// TwinCAT 3 PLC project XtsLib
// Title: Xts Library
// Company: BeckhoffUK
// Author: ChrisK
// ProjectVersion: 1.0.0.6
// Description: Xts framework implementation
// ProgramVersion: 3.1.4023.0
// libraries:
//   Tc2_Standard, * (Beckhoff Automation GmbH)
//   Tc2_System, * (Beckhoff Automation GmbH)
//   Tc3_EventLogger, * (Beckhoff Automation GmbH)
//   Tc3_McCoordinatedMotion, * (Beckhoff Automation GmbH)
//   Tc3_Module, * (Beckhoff Automation GmbH)
//   Tc3_PackML_V2, * (Beckhoff Automation GmbH)
//   Tc3_XTS_Utility, * (Beckhoff Automation GmbH)
//   Tc2_MC2,newest,Beckhoff Automation GmbH
//   Tc3_Mc3Definitions,newest,Beckhoff Automation GmbH
//   Tc3_McCollisionAvoidance,newest,Beckhoff Automation GmbH
// project tree:
//   Axis Class/ MC2_Axis_Base.TcPOU
//   EventLoggerClass/ ITcMessage_Ext.TcIO, TcMessage_Ext.TcPOU
//   Mover Class/ FB_Mover.TcPOU, GearMover.TcPOU, IDynamics.TcIO, IGearMover.TcIO, IMover.TcIO, ITmsMover.TcIO, TMS_Mover.TcPOU
//   PackML/ IPmlStateMachine.TcIO, PMLStateMachine.TcPOU
//   PackML_Method_Pattern/ PML_Method_Base.TcPOU
//   SequenceSamples/ GearMoverSequence.TcPOU (not stored), IndexMoverSequence.TcPOU, IndexSequenceState.TcDUT, MoverSequenceInfo.TcDUT
//   Station Class/Process/ IProcess.TcIO, Process.TcPOU
//   Station Class/Station/ IStation.TcIO, Station.TcPOU, StationSample.TcPOU, stStationInfo.TcDUT, stStationStatus.TcDUT
//   Station Class/TMSStation/ ITF_SwitchStation.TcIO, TmsEmbarkStation.TcPOU, TmsExchange.TcPOU, TmsHoldStation.TcPOU
//   Switch Class/ DualModuleTmsSwitch.TcPOU, ITF_TmsSwitch.TcIO, TmsSwitchPosition.TcDUT, TmsSwitchInfo.TcDUT, TmsSwitchMode.TcDUT, TmsSwitchState.TcDUT
//   / SystemParameters.TcGVL
//   Tasks/ ActivateTrackForMover.TcPOU, AddMoverToGroupTask.TcPOU, AxesReset.TcPOU, DisableGroup.TcPOU, EnableGroup.TcPOU, GearInCA.TcPOU, HaltMover.TcPOU, Mc2Halt.TcPOU, ITask.TcIO, Mc2MoveToPosition.TcPOU, MoveModuloMoverToPosition.TcPOU, MoveMoverToPosition.TcPOU, MoveMoverToPositionZoned.TcPOU, RemoveAllMoverFromGroup.TcPOU, ResetGroup.TcPOU, StopMoverGroup.TcPOU, XtsDisableSequence.TcPOU, XtsEnableSequence.TcPOU
//   XTS Class/ ITF_StartUpSequence.TcIO, IXtsTrack.TcIO, XtsTrack.TcPOU
//   XTS Class/Xts Collision Group/ CAGroupInfo.TcDUT (not stored), CAGroupStatus.TcDUT (not stored), CollisionGroup.TcPOU, ICollisionGroup.TcIO (not stored)
//   XTS Class/Xts Hardware/ XtsHardware.TcPOU, XtsHardwareInfo.TcDUT, XtsHardwareState.TcDUT

// ---- SequenceSamples/IndexSequenceState.TcDUT
{attribute 'qualified_only'}
{attribute 'strict'}
TYPE IndexSequenceState :
(
	Init := 0,                                               
	Available := 1,
	MovingToStart := 2, 
	AtStart := 3,                                 
	MovingToStation := 4,
	QueuedAtStation := 5,
	AtStation := 6,
	AtProcess := 7,
	InProcess := 8,
	GetNextMove := 9,
	GoToNextStation := 10,
	Stopping := 11,
	Aborting := 12
);
END_TYPE

// ---- SequenceSamples/MoverSequenceInfo.TcDUT
TYPE MoverSequenceInfo :
STRUCT
	MoverId : UDINT;
	CurrentStation : INT;
	Velocity : MC_LREAL;
	State : IndexSequenceState;
END_STRUCT
END_TYPE

// ---- Station Class/Station/stStationInfo.TcDUT
TYPE stStationInfo :
STRUCT
	StationProcessTime : TIME;
	StationPosition : MC_LREAL;
	StationStatus : stStationStatus;
END_STRUCT
END_TYPE

// ---- Station Class/Station/stStationStatus.TcDUT
TYPE stStationStatus :
STRUCT
	Clear : BOOL;
	Complete : BOOL;
	Operating : BOOL;
	Ready : BOOL;
	HasMover : BOOL;
END_STRUCT
END_TYPE

// ---- Switch Class/TmsSwitchPosition.TcDUT
{attribute 'qualified_only'}
{attribute 'strict'}
TYPE TmsSwitchPosition :
(
	Up := 0,
	Middle := 1,
	Down := 2,
	Moving := 3
);
END_TYPE

// ---- Switch Class/TmsSwitchInfo.TcDUT
TYPE TmsSwitchInfo :
STRUCT
	State : TmsSwitchState;
	Mode : TmsSwitchMode;
	Position : TmsSwitchPosition;
	ActPos : MC_LREAL;
END_STRUCT
END_TYPE

// ---- Switch Class/TmsSwitchMode.TcDUT
{attribute 'qualified_only'}
{attribute 'strict'}
TYPE TmsSwitchMode :
(
	Automatic := 0,
	Manual := 1
);
END_TYPE

// ---- Switch Class/TmsSwitchState.TcDUT
{attribute 'qualified_only'}
{attribute 'strict'}
TYPE TmsSwitchState :
(
	Init := 0,                                               
	Ready := 1,                                 
	Enabling := 2,
	Enabled := 3,
	Resetting := 4,
	Waiting := 5,
	AssignMover := 6,
	Moving := 7,
	Done := 8,
	Disabling := 9
);
END_TYPE

// ---- XTS Class/Xts Hardware/XtsHardwareInfo.TcDUT
TYPE XtsHardwareInfo :
STRUCT
	NoOfParts: UDINT;
	NoOfTracks : UDINT;
	NoOfModules : ARRAY[1..10] OF UDINT;
	HWState : XtsHardwareState;
END_STRUCT
END_TYPE

// ---- XTS Class/Xts Hardware/XtsHardwareState.TcDUT
{attribute 'qualified_only'}
{attribute 'strict'}
TYPE XtsHardwareState :
(
	Init := 0,
	SetDetection := 1,                                               
	Redetect := 2,
	MoversValid := 3,                                 
	AllMoversFound := 4,
	MoverIdDetection := 5,
	XTSMode := 6,
	CheckModuleVoltages := 7,
	HWReady := 8
);
END_TYPE

// ---- SystemParameters.TcGVL
{attribute 'qualified_only'}
VAR_GLOBAL CONSTANT
	nModuleNumber  : UINT := 16;
	NumberOfMovers : INT := 10;
	NumberOfStations : INT := 6;
	TrackLength : LREAL := 4000.0;
	TrackHomePosition : LREAL := 800.0;
	Tracks : UDINT := 1;
END_VAR

// ---- EventLoggerClass/ITcMessage_Ext.TcIO
INTERFACE ITcMessage_Ext

METHOD Send : BOOL
VAR_INPUT
	eventType : Tc3_EventLogger.TcEventEntry;
	args : STRING(255);
END_VAR
END_METHOD

END_INTERFACE

// ---- Mover Class/IDynamics.TcIO
INTERFACE IDynamics

PROPERTY Acceleration : mc_lreal
GET
END_GET
SET
END_SET
END_PROPERTY

PROPERTY Deceleration : mc_lreal
GET
END_GET
SET
END_SET
END_PROPERTY

PROPERTY Jerk : mc_lreal
GET
END_GET
SET
END_SET
END_PROPERTY

END_INTERFACE

// ---- Mover Class/IGearMover.TcIO
INTERFACE IGearMover EXTENDS IMover

METHOD Gear : BOOL
VAR_INPUT
	MasterPosition : MC_LREAL;
	SlavePosition : MC_LREAL;
END_VAR
END_METHOD

METHOD inGear : BOOL
VAR_INPUT
END_VAR
END_METHOD

METHOD isMaster : BOOL
VAR_INPUT
END_VAR
END_METHOD

METHOD masterAxis : UDINT
VAR_INPUT
END_VAR
END_METHOD

END_INTERFACE

// ---- Mover Class/IMover.TcIO
INTERFACE IMover EXTENDS __SYSTEM.IQueryInterface

PROPERTY AxisRef : reference to axis_ref
GET
END_GET
END_PROPERTY

METHOD DisableAxis : BOOL
VAR_INPUT
END_VAR
END_METHOD

METHOD EnableAxis : BOOL
VAR_INPUT
END_VAR
END_METHOD

METHOD HaltAxis : BOOL
VAR_INPUT
END_VAR
END_METHOD

METHOD HasCommand : BOOL
VAR_INPUT
END_VAR
END_METHOD

METHOD hasError : BOOL
VAR_INPUT
END_VAR
END_METHOD

PROPERTY IdentInGroup : int
GET
END_GET
SET
END_SET
END_PROPERTY

METHOD isAtPosition : BOOL
VAR_INPUT
	position : MC_LREAL;
END_VAR
END_METHOD

METHOD isDetected : BOOL
VAR_INPUT
END_VAR
END_METHOD

METHOD isEnabled : BOOL
VAR_INPUT
END_VAR
END_METHOD

METHOD isPastPosition : BOOL
VAR_INPUT
	position : MC_LREAL;
END_VAR
END_METHOD

METHOD isStationary : BOOL
VAR_INPUT
END_VAR
END_METHOD

METHOD MoveTo : BOOL
VAR_INPUT
	Position : MC_LREAL;
	Velocity : MC_LREAL;
	BackwardMove : BOOL;
END_VAR
END_METHOD

METHOD ResetAxis : BOOL
VAR_INPUT
END_VAR
END_METHOD

END_INTERFACE

// ---- Mover Class/ITmsMover.TcIO
INTERFACE ITmsMover EXTENDS IMover

METHOD ActivateTrack : BOOL
VAR_INPUT
	newTrack : OTCID;
END_VAR
END_METHOD

PROPERTY ActiveTrack : OTCID
GET
END_GET
END_PROPERTY

METHOD SetMoverInterface : BOOL
VAR_INPUT
	MoverInterface : I_TcIoXtsXpuMover;
END_VAR
END_METHOD

END_INTERFACE

// ---- PackML/IPmlStateMachine.TcIO
INTERFACE IPmlStateMachine

METHOD public GetCurrentMode : E_PmlProtectedUnitMode
VAR_INPUT
END_VAR
END_METHOD

METHOD GetCurrentState : E_PMLState
VAR_INPUT
END_VAR
END_METHOD

METHOD PmlModeCommand : BOOL
VAR_INPUT
	Mode : E_PMLProtectedUnitMode;
END_VAR
END_METHOD

METHOD PmlStateCommand : bool
VAR_INPUT
	Command : E_PMLCommand;
END_VAR
END_METHOD

METHOD SetStateComplete : BOOL
VAR_INPUT
END_VAR
END_METHOD

END_INTERFACE

// ---- Station Class/Process/IProcess.TcIO
INTERFACE IProcess EXTENDS IStation

PROPERTY EndPosition : MC_LREAL
GET
END_GET
SET
END_SET
END_PROPERTY

PROPERTY IsProcess : booL
GET
END_GET
SET
END_SET
END_PROPERTY

PROPERTY ProcessVelocity : mc_lreal
GET
END_GET
SET
END_SET
END_PROPERTY

PROPERTY StartPosition : MC_LREAL
GET
END_GET
SET
END_SET
END_PROPERTY

END_INTERFACE

// ---- Station Class/Station/IStation.TcIO
INTERFACE IStation

METHOD Abort : BOOL
VAR_INPUT
END_VAR
END_METHOD

METHOD HasMover : BOOL
VAR_INPUT
	mover : IMover;
END_VAR
END_METHOD

METHOD IsClear : BOOL
VAR_INPUT
END_VAR
END_METHOD

METHOD isComplete : BOOL
VAR_INPUT
END_VAR
END_METHOD

PROPERTY IsLastStation : BOOL
GET
END_GET
SET
END_SET
END_PROPERTY

METHOD IsOperating : BOOL
VAR_INPUT
END_VAR
END_METHOD

METHOD IsReady : BOOL
VAR_INPUT
END_VAR
END_METHOD

METHOD MoverAway : BOOL
VAR_INPUT
END_VAR
END_METHOD

PROPERTY Position : MC_LREAL
GET
END_GET
SET
END_SET
END_PROPERTY

END_INTERFACE

// ---- Station Class/TMSStation/ITF_SwitchStation.TcIO
INTERFACE ITF_SwitchStation EXTENDS __SYSTEM.IQueryInterface

PROPERTY StationPosition : int
GET
END_GET
SET
END_SET
END_PROPERTY

METHOD SwitchMoveComplete : BOOL
VAR_INPUT
END_VAR
END_METHOD

PROPERTY SwitchPosition : mc_lreal
GET
END_GET
SET
END_SET
END_PROPERTY

END_INTERFACE

// ---- Switch Class/ITF_TmsSwitch.TcIO
INTERFACE ITF_TmsSwitch

METHOD ExchangeMover : BOOL
VAR_INPUT
	Mover : IMover;
	currentStation : ITF_SwitchStation;
END_VAR
END_METHOD

METHOD HasMover : BOOL
VAR_INPUT
END_VAR
END_METHOD

METHOD IsStationary : BOOL
VAR_INPUT
END_VAR
END_METHOD

METHOD MoveTo : BOOL
VAR_INPUT
	positionState : TmsSwitchPosition;
END_VAR
END_METHOD

PROPERTY Switch : TmsSwitchPosition
GET
END_GET
END_PROPERTY

END_INTERFACE

// ---- Tasks/ITask.TcIO
INTERFACE ITask

METHOD Abort : BOOL
VAR_INPUT
END_VAR
END_METHOD

PROPERTY Busy : bool
GET
END_GET
END_PROPERTY

PROPERTY Done : bool
GET
END_GET
END_PROPERTY

PROPERTY Error : bool
GET
END_GET
END_PROPERTY

END_INTERFACE

// ---- XTS Class/ITF_StartUpSequence.TcIO
INTERFACE ITF_StartUpSequence

METHOD Call : BOOL
VAR_INPUT
END_VAR
END_METHOD

END_INTERFACE

// ---- XTS Class/IXtsTrack.TcIO
INTERFACE IXtsTrack

PROPERTY HomePosition : MC_LREAL
GET
END_GET
SET
END_SET
END_PROPERTY

PROPERTY TrackLength : mc_lreal
GET
END_GET
SET
END_SET
END_PROPERTY

END_INTERFACE

// ---- Axis Class/MC2_Axis_Base.TcPOU
FUNCTION_BLOCK MC2_Axis_Base EXTENDS CyclicBase
VAR_INPUT
END_VAR
VAR_OUTPUT
END_VAR
VAR
	_axis : Tc2_MC2.AXIS_REF;
	axesEnable		: AxisPower(_axis);
	axesReset		: AxesReset(_axis);
	axesMoveTo 		: Mc2MoveToPosition(_axis);
	axesHalt 		: Mc2Halt(_axis);
	axesReadError : Tc2_MC2.MC_ReadAxisError;
	_MoverErrorId: DWORD;
END_VAR

METHOD Cycle : BOOL
VAR_INPUT
END_VAR
axesMoveTo.Cycle();
axesHalt.Cycle();
axesReset.Cycle();
_axis.ReadStatus();
axesEnable.Cycle();
axesReadError(Axis := _axis, Enable := TRUE, AxisErrorID => _MoverErrorId);
END_METHOD

METHOD PUBLIC DisableAxis : BOOL
VAR_INPUT
END_VAR
DisableAxis := axesEnable.Disable();
END_METHOD

METHOD PUBLIC EnableAxis : BOOL
VAR_INPUT
END_VAR
EnableAxis := axesEnable.Enable();
END_METHOD

METHOD PUBLIC HaltAxis : BOOL
VAR_INPUT
END_VAR
IF NOT axesHalt.Busy THEN
	axesHalt.Execute();
	axesMoveTo.Abort();
	HaltAxis := TRUE;
END_IF
END_METHOD

METHOD hasError : BOOL
VAR_INPUT
END_VAR
hasError := _axis.Status.Error;
END_METHOD

METHOD isAtPosition : BOOL
VAR_INPUT
	position : MC_LREAL;
END_VAR
IF _axis.NcToPlc.ActPos < position + 0.2 AND _axis.NcToPlc.ActPos > position - 0.2 THEN
	isAtPosition := TRUE;
END_IF
END_METHOD

METHOD isEnabled : BOOL
VAR_INPUT
END_VAR
isEnabled := not _axis.Status.Disabled;
END_METHOD

METHOD PUBLIC isStationary : BOOL
VAR_INPUT
END_VAR
isStationary := _axis.NcToPlc.SetVelo = 0;
END_METHOD

METHOD PUBLIC MoveToPosition : BOOL
VAR_INPUT
	Position : MC_LREAL;
	Velocity : MC_LREAL;
END_VAR
IF NOT isAtPosition(position := Position) THEN
	IF NOT axesMoveTo.Busy THEN
		axesMoveTo.MoveTo(Position := Position, Velocity := Velocity);
		MoveToPosition := TRUE;
	END_IF
END_IF
END_METHOD

METHOD PUBLIC ResetAxis : BOOL
VAR_INPUT
END_VAR
axesReset.Execute();
axesMoveTo.Abort();
axesHalt.Abort();
END_METHOD

END_FUNCTION_BLOCK

// ---- Tasks/AxesReset.TcPOU
{attribute 'hide_all_locals'}
FUNCTION_BLOCK AxesReset EXTENDS TaskBase
VAR_INPUT
END_VAR
VAR_OUTPUT
END_VAR
VAR
	resetMover : Tc2_MC2.MC_Reset;
	_axis : REFERENCE TO Tc2_MC2.AXIS_REF;
	_ResetMover : BOOL;
END_VAR

METHOD Abort : BOOL
resetMover.Execute := FALSE;
_busy := FALSE;
_ResetMover := FALSE;
Abort := TRUE;
State := 0;
END_METHOD

METHOD Cycle : BOOL
VAR_INPUT
END_VAR
CASE State OF
	0:
		IF _ResetMover THEN
			_done := FALSE;
			_error := FALSE;
			_busy := TRUE;
			resetMover.Execute := TRUE;
			IF resetMover.Busy THEN
				State := 10;
				_ResetMover := FALSE;
			END_IF
		END_IF
	
	10:
		IF NOT resetMover.Busy THEN
			IF resetMover.Done THEN
				_done := TRUE;
			ELSIF resetMover.Error THEN
				_error := TRUE;
			END_IF
			_busy := FALSE;
			resetMover.Execute := FALSE;
			State := 0;
		END_IF
END_CASE

resetMover(Axis := _axis);
END_METHOD

METHOD Execute : BOOL
VAR_INPUT
END_VAR
Execute := _ResetMover := true;
END_METHOD

METHOD FB_init : BOOL
VAR_INPUT
	bInitRetains : BOOL; // if TRUE, the retain variables are initialized (warm start / cold start)
	bInCopyCode : BOOL;  // if TRUE, the instance afterwards gets moved into the copy code (online change)
	axis : reference TO AXIS_REF;
END_VAR
_axis REF= axis;
END_METHOD

END_FUNCTION_BLOCK

// ---- Tasks/Mc2MoveToPosition.TcPOU
FUNCTION_BLOCK Mc2MoveToPosition EXTENDS TaskBase
VAR_INPUT
END_VAR
VAR_OUTPUT
END_VAR
VAR
	moveAbs	: MC_MoveAbsolute;
	_axis : REFERENCE TO AXIS_REF;
	_MoveSwitch : BOOL;
END_VAR

METHOD Abort : BOOL
moveAbs.Execute := FALSE;
moveAbs.Position := moveAbs.Velocity := 0;
_MoveSwitch := false;
_busy := false;
Abort := true;
State := 0;
END_METHOD

PROPERTY PUBLIC Acceleration : mc_lreal
GET
Acceleration := moveAbs.Acceleration;
END_GET
SET
moveAbs.Acceleration := Acceleration;
END_SET
END_PROPERTY

METHOD Cycle : BOOL
VAR_INPUT
END_VAR
CASE State OF
	0:
		IF _MoveSwitch THEN
			_done := FALSE;
			_error := FALSE;
			_busy := TRUE;
			moveAbs.Execute := TRUE;
			IF moveAbs.Busy THEN
				State := 10;
				_MoveSwitch := FALSE;
			END_IF
		END_IF
		
	10:
		IF NOT moveAbs.Busy THEN
			IF moveAbs.Done THEN
				_done := TRUE;
			ELSIF moveAbs.Error THEN
				_error := TRUE;
			END_IF
			_busy := FALSE;
			moveAbs.Execute := FALSE;
			State := 0;
		END_IF
END_CASE

moveAbs(Axis := _axis);
END_METHOD

PROPERTY PUBLIC Deceleration : mc_lreal
GET
Deceleration := moveAbs.Deceleration;
END_GET
SET
moveAbs.Deceleration := Deceleration;
END_SET
END_PROPERTY

METHOD FB_init : BOOL
VAR_INPUT
	bInitRetains : BOOL; // if TRUE, the retain variables are initialized (warm start / cold start)
	bInCopyCode : BOOL;  // if TRUE, the instance afterwards gets moved into the copy code (online change)
	axis : reference TO AXIS_REF;
END_VAR
_axis REF= axis;
END_METHOD

PROPERTY PUBLIC Jerk : mc_lreal
GET
Jerk := moveAbs.Jerk;
END_GET
SET
moveAbs.Jerk := Jerk;
END_SET
END_PROPERTY

METHOD MoveTo : BOOL
VAR_INPUT
	Position : MC_LREAL;
	Velocity : MC_LREAL;
END_VAR
moveAbs.Position := Position;
moveAbs.Velocity := Velocity;
_MoveSwitch := MoveTo := true;
END_METHOD

END_FUNCTION_BLOCK

// ---- Tasks/Mc2Halt.TcPOU
{attribute 'hide_all_locals'}
FUNCTION_BLOCK Mc2Halt EXTENDS TaskBase
VAR_INPUT
END_VAR
VAR_OUTPUT
END_VAR
VAR
	mcHalt : Tc2_MC2.MC_Halt;
	_axis : REFERENCE TO Tc2_MC2.AXIS_REF;
	_Halt : BOOL;
END_VAR

METHOD Abort : BOOL
mchalt.Execute := FALSE;
_busy := FALSE;
_Halt := FALSE;
Abort := TRUE;
State := 0;
END_METHOD

METHOD Cycle : BOOL
VAR_INPUT
END_VAR
CASE State OF
	0:
		IF _Halt THEN
			_done := FALSE;
			_error := FALSE;
			_busy := TRUE;
			mcHalt.Execute := TRUE;
			IF mcHalt.Busy THEN
				State := 10;
				_Halt := FALSE;
			END_IF
		END_IF
	
	10:
		IF NOT mcHalt.Busy THEN
			IF mcHalt.Done THEN
				_done := TRUE;
			ELSIF mcHalt.Error THEN
				_error := TRUE;
			END_IF
			_busy := FALSE;
			mcHalt.Execute := FALSE;
			State := 0;
		END_IF
END_CASE

mcHalt(Axis := _axis);
END_METHOD

METHOD Execute : BOOL
VAR_INPUT
END_VAR
Execute := _Halt := true;
END_METHOD

METHOD FB_init : BOOL
VAR_INPUT
	bInitRetains : BOOL; // if TRUE, the retain variables are initialized (warm start / cold start)
	bInCopyCode : BOOL;  // if TRUE, the instance afterwards gets moved into the copy code (online change)
	axis : reference TO AXIS_REF;
END_VAR
_axis REF= axis;
END_METHOD

END_FUNCTION_BLOCK

// ---- EventLoggerClass/TcMessage_Ext.TcPOU
FUNCTION_BLOCK TcMessage_Ext IMPLEMENTS ITcMessage_Ext
VAR_INPUT
END_VAR
VAR_OUTPUT
END_VAR
VAR
    fbMsg : FB_TcMessage; 
	_loggerLevel : TcEventSeverity := TcEventSeverity.Info;
END_VAR

PROPERTY PUBLIC LoggerLevel : TcEventSeverity
GET
LoggerLevel := _loggerLevel;
END_GET
SET
_loggerLevel := LoggerLevel;
END_SET
END_PROPERTY

METHOD PUBLIC Send : BOOL
VAR_INPUT
	eventType : Tc3_EventLogger.TcEventEntry;
	args : STRING(255);
END_VAR
IF eventType.eSeverity >= LoggerLevel THEN
	THIS^.fbMsg.CreateEx(eventType, 0);
	THIS^.fbMsg.ipArguments.AddString(args);
	THIS^.fbMsg.Send(0);
	THIS^.fbMsg.Release();
END_IF
END_METHOD

END_FUNCTION_BLOCK

// ---- Mover Class/FB_Mover.TcPOU
FUNCTION_BLOCK FB_Mover EXTENDS CyclicBase IMPLEMENTS IMover, IDynamics
VAR
	axesEnable		: AxisPower(_axis);
	axesReset		: AxesReset(_axis);
	axesMoveTo 		: MoveMoverToPosition(_axis) := (Gap := 100.0);
	axesHalt 		: HaltMover(_axis);
	axesReadError : Tc2_MC2.MC_ReadAxisError;
	_axis 			: AXIS_REF;
	_identInGroup : INT;
	_trackLength : MC_LREAL;
	_targetPos : LREAL;
	_MoverErrorId : DWORD;
	_arrZones : ARRAY[1..4] OF DINT;
	_arrVelocities : ARRAY[1..4] OF mc_LREAL;
END_VAR

PROPERTY PUBLIC Acceleration : mc_lreal
GET
Acceleration := axesMoveTo.Acceleration;
END_GET
SET
axesMoveTo.Acceleration := Acceleration;
END_SET
END_PROPERTY

PROPERTY PUBLIC AxisRef : reference to AXIS_REF
GET
AxisRef REF= THIS^._axis;
END_GET
END_PROPERTY

METHOD PUBLIC  Cycle : BOOL
VAR_INPUT
END_VAR
axesMoveTo.Cycle();
axesHalt.Cycle();
axesReset.Cycle();
_axis.ReadStatus();
axesEnable.Cycle();
axesReadError(Axis := _axis, Enable := TRUE, AxisErrorID => _MoverErrorId);
END_METHOD

PROPERTY PUBLIC Deceleration : mc_lreal
GET
Deceleration := axesMoveTo.Deceleration;
END_GET
SET
axesMoveTo.Deceleration := Deceleration;
END_SET
END_PROPERTY

METHOD PUBLIC DisableAxis : BOOL
VAR_INPUT
END_VAR
DisableAxis := axesEnable.Disable();
END_METHOD

METHOD PUBLIC EnableAxis : BOOL
VAR_INPUT
END_VAR
EnableAxis := axesEnable.Enable();
END_METHOD

PROPERTY PUBLIC Gap : mc_lreal
GET
Gap := axesMoveTo.Gap;
END_GET
SET
axesMoveTo.Gap := Gap;
END_SET
END_PROPERTY

METHOD PUBLIC HaltAxis : BOOL
VAR_INPUT
END_VAR
IF NOT axesHalt.Busy THEN
	axesHalt.Execute();
	HaltAxis := TRUE;
	axesMoveTo.Abort();
END_IF
END_METHOD

METHOD PUBLIC HasCommand : BOOL
VAR_INPUT
END_VAR
HasCommand := axesMoveTo.Busy;
END_METHOD

METHOD hasError : BOOL
VAR_INPUT
END_VAR
hasError := _axis.Status.Error;
END_METHOD

PROPERTY PUBLIC IdentInGroup : int
GET
IdentInGroup := _identInGroup;
END_GET
SET
_identInGroup := IdentInGroup;
END_SET
END_PROPERTY

METHOD isAtPosition : BOOL
VAR_INPUT
	position : MC_LREAL;
END_VAR
IF position > 1 THEN
	IF _axis.NcToPlc.ModuloActPos < position + 1 AND _axis.NcToPlc.ModuloActPos > position - 1 THEN
		isAtPosition := TRUE;
	END_IF  
ELSE
	IF _axis.NcToPlc.ModuloActPos < position + 1 AND _axis.NcToPlc.ModuloActPos > 0.0  
		OR _axis.NcToPlc.ModuloActPos < _trackLength AND _axis.NcToPlc.ModuloActPos > _trackLength - 1 THEN
		isAtPosition := TRUE;
	END_IF
END_IF
END_METHOD

METHOD PUBLIC isDetected : BOOL
VAR_INPUT
END_VAR
IF _axis.NcToPlc.AxisId = 0 THEN
	RETURN;
END_IF
isDetected := true;
END_METHOD

METHOD isEnabled : BOOL
VAR_INPUT
END_VAR
isEnabled := not _axis.Status.Disabled;
END_METHOD

METHOD PUBLIC isPastPosition : BOOL
VAR_INPUT
	position : MC_LREAL;
END_VAR
IF position > 1 THEN
	IF _axis.NcToPlc.ModuloActPos > position THEN
		isPastPosition := TRUE;
	END_IF  
END_IF
END_METHOD

METHOD PUBLIC isStationary : BOOL
VAR_INPUT
END_VAR
isStationary := _axis.NcToPlc.SetVelo = 0;
END_METHOD

PROPERTY PUBLIC Jerk : mc_lreal
GET
Jerk := axesMoveTo.Jerk;
END_GET
SET
axesMoveTo.Jerk := Jerk;
END_SET
END_PROPERTY

METHOD PROTECTED ModuloToAbs : mc_lreal
VAR_INPUT
	moduloPositionDemand: MC_LREAL;
	_backwardsAllowed : BOOL;
END_VAR
//---------code to set actual position from modulo command----------------------
IF NOT _backwardsAllowed THEN
	//--------if you want to go forward-------------------------------------------------------------
	//---------if SetPos is greater than current actual then move to that position--------------------
	//---------else current position is greater, increase moduloturn count by 1 before set---------------
	IF moduloPositionDemand > _axis.NcToPlc.ModuloActPos THEN
		ModuloToAbs := (DINT_TO_LREAL(_Axis.NcToPlc.ModuloActTurns)*_trackLength) + moduloPositionDemand;
	ELSE
		ModuloToAbs := (DINT_TO_LREAL(_Axis.NcToPlc.ModuloActTurns + 1)*_trackLength) + moduloPositionDemand;
	END_IF
ELSE
	//--------if you want to go backwards--------------------------------
	//--------if setPos is less than current actual then move to that position---------------------
	//---------else current position is less, decrease moduloturn count by 1 before set------------
	IF moduloPositionDemand < _axis.NcToPlc.ModuloActPos THEN
		ModuloToAbs := (DINT_TO_LREAL(_Axis.NcToPlc.ModuloActTurns)*_trackLength) + moduloPositionDemand;
	ELSE
		ModuloToAbs := (DINT_TO_LREAL(_Axis.NcToPlc.ModuloActTurns-1)*_trackLength) + moduloPositionDemand;
	END_IF
END_IF
END_METHOD

PROPERTY MoverErrorId : dword
GET
MoverErrorId := _MoverErrorId;
END_GET
SET
_MoverErrorId := MoverErrorId;
END_SET
END_PROPERTY

METHOD PUBLIC MoveTo : BOOL
VAR_INPUT
	Position : MC_LREAL;
	Velocity : MC_LREAL;
	BackwardMove : BOOL;
END_VAR
IF NOT isAtPosition(position := Position) THEN
	IF NOT axesMoveTo.Busy THEN
		axesMoveTo.MoveTo(Position := ModuloToAbs(Position, BackwardMove), Velocity := Velocity);
		MoveTo := TRUE;
		_targetPos := Position;
	END_IF
END_IF
END_METHOD

METHOD PUBLIC ResetAxis : BOOL
VAR_INPUT
END_VAR
VAR
END_VAR
axesReset.Execute();
axesMoveTo.Abort();
axesHalt.Abort();
END_METHOD

PROPERTY PUBLIC TrackLength : MC_LREAL
GET
TrackLength := _trackLength;
END_GET
SET
_trackLength := TrackLength;
END_SET
END_PROPERTY

PROPERTY Zones : array[1..4] of dint
GET
Zones := _arrZones;
END_GET
SET
_arrZones := Zones;
END_SET
END_PROPERTY

PROPERTY ZoneVelocities : array[1..4] of mc_lreal
GET
ZoneVelocities := _arrVelocities;
END_GET
SET
_arrVelocities := ZoneVelocities;
END_SET
END_PROPERTY

END_FUNCTION_BLOCK

// ---- Tasks/MoveMoverToPosition.TcPOU
FUNCTION_BLOCK MoveMoverToPosition EXTENDS TaskBase
VAR_INPUT
END_VAR
VAR_OUTPUT
END_VAR
VAR
	moveAbs	: MC_MoveAbsoluteCA;
	_axis : REFERENCE TO AXIS_REF;
	_MoveMover : BOOL;
	_stOptions : ST_MoveAbsoluteCAOptions;
END_VAR

METHOD Abort : BOOL
moveAbs.Execute := FALSE;
moveAbs.Position := moveAbs.Velocity := 0;
_MoveMover := false;
_busy := false;
Abort := true;
State := 0;
END_METHOD

PROPERTY PUBLIC Acceleration : mc_lreal
GET
Acceleration := moveAbs.Acceleration;
END_GET
SET
moveAbs.Acceleration := Acceleration;
END_SET
END_PROPERTY

METHOD Cycle : BOOL
VAR_INPUT
END_VAR
CASE State OF
	0:
		IF _MoveMover THEN
			_done := FALSE;
			_error := FALSE;
			_busy := TRUE;
			moveAbs.Execute := TRUE;
			IF moveAbs.Busy THEN
				State := 10;
				_MoveMover := FALSE;
			END_IF
		END_IF
		
	10:
		IF NOT moveAbs.Busy THEN
			IF moveAbs.Done THEN
				_done := TRUE;
			ELSIF moveAbs.Error THEN
				_error := TRUE;
			END_IF
			_busy := FALSE;
			moveAbs.Execute := FALSE;
			State := 0;
		END_IF
END_CASE

moveAbs(Axis := _axis, Options := _stOptions);
END_METHOD

PROPERTY PUBLIC Deceleration : mc_lreal
GET
Deceleration := moveAbs.Deceleration;
END_GET
SET
moveAbs.Deceleration := Deceleration;
END_SET
END_PROPERTY

METHOD FB_init : BOOL
VAR_INPUT
	bInitRetains : BOOL; // if TRUE, the retain variables are initialized (warm start / cold start)
	bInCopyCode : BOOL;  // if TRUE, the instance afterwards gets moved into the copy code (online change)
	axis : reference TO AXIS_REF;
END_VAR
_axis REF= axis;
END_METHOD

PROPERTY PUBLIC Gap : mc_lreal
GET
Gap := moveAbs.Gap;
END_GET
SET
moveAbs.Gap := Gap;
END_SET
END_PROPERTY

PROPERTY PUBLIC Jerk : mc_lreal
GET
Jerk := moveAbs.Jerk;
END_GET
SET
moveAbs.Jerk := Jerk;
END_SET
END_PROPERTY

METHOD MoveTo : BOOL
VAR_INPUT
	Position : MC_LREAL;
	Velocity : MC_LREAL;
END_VAR
moveAbs.Position := Position;
moveAbs.Velocity := Velocity;
_MoveMover := MoveTo := true;
END_METHOD

PROPERTY PUBLIC Options : ST_MoveAbsoluteCAOptions
GET
Options := _stOptions;
END_GET
SET
_stOptions := Options;
END_SET
END_PROPERTY

END_FUNCTION_BLOCK

// ---- Tasks/HaltMover.TcPOU
{attribute 'hide_all_locals'}
FUNCTION_BLOCK HaltMover EXTENDS TaskBase
VAR_INPUT
END_VAR
VAR_OUTPUT
END_VAR
VAR
	haltMover : Tc3_McCollisionAvoidance.MC_HaltCA;
	_axis : REFERENCE TO Tc2_MC2.AXIS_REF;
	_HaltMover : BOOL;
END_VAR

METHOD Abort : BOOL
haltMover.Execute := FALSE;
_busy := FALSE;
_HaltMover := FALSE;
Abort := TRUE;
State := 0;
END_METHOD

METHOD Cycle : BOOL
VAR_INPUT
END_VAR
CASE State OF
	0:
		IF _HaltMover THEN
			_done := FALSE;
			_error := FALSE;
			_busy := TRUE;
			haltMover.Execute := TRUE;
			IF haltMover.Busy THEN
				State := 10;
				_HaltMover := FALSE;
			END_IF
		END_IF
	
	10:
		IF NOT haltMover.Busy THEN
			IF haltMover.Done THEN
				_done := TRUE;
			ELSIF haltMover.Error THEN
				_error := TRUE;
			END_IF
			_busy := FALSE;
			haltMover.Execute := FALSE;
			State := 0;
		END_IF
END_CASE

haltMover(Axis := _axis);
END_METHOD

METHOD Execute : BOOL
VAR_INPUT
END_VAR
Execute := _HaltMover := true;
END_METHOD

METHOD FB_init : BOOL
VAR_INPUT
	bInitRetains : BOOL; // if TRUE, the retain variables are initialized (warm start / cold start)
	bInCopyCode : BOOL;  // if TRUE, the instance afterwards gets moved into the copy code (online change)
	axis : reference TO AXIS_REF;
END_VAR
_axis REF= axis;
END_METHOD

END_FUNCTION_BLOCK

// ---- Mover Class/GearMover.TcPOU
FUNCTION_BLOCK GearMover EXTENDS FB_Mover IMPLEMENTS IGearMover
VAR_INPUT
	XtsTrack : IXtsTrack;
	StateMachine : IPmlStateMachine;
END_VAR
VAR_OUTPUT
END_VAR
VAR
	moverSequence : GearMoverSequence;
	bInit : BOOL;
	CurrentLimit AT%Q* : INT;
	Mode AT%Q* : UINT;
	axesGear	: GearInCA;
	isMasterAxis: BOOL;
	MoverToGearTo: UDINT := 1;
END_VAR
VAR_IN_OUT
	MoverArray : ARRAY[*] OF IGearMover;
END_VAR

METHOD PUBLIC  Cycle : BOOL
VAR_INPUT
END_VAR
IF NOT bInit THEN
	IF THIS^._axis.NcToPlc.AxisId <> 0 THEN
		IF (THIS^._axis.NcToPlc.AxisId MOD 2)<>1 THEN
			Mode.8 := TRUE;
			isMasterAxis := TRUE;
		ELSE
			isMasterAxis := FALSE;
			MoverToGearTo := THIS^.AxisRef.NcToPlc.AxisId + 1;
		END_IF
		bInit := TRUE;
	END_IF
END_IF
	_trackLength := XtsTrack.TrackLength;
IF isMasterAxis THEN
	IF (_axis.NcToPlc.ModuloActPos > 3400 OR _axis.NcToPlc.ModuloActPos < 300)  THEN
		CurrentLimit := 1000;
	ELSE
		CurrentLimit := 2000;
	END_IF
ELSE
	CurrentLimit := 12000;
END_IF

SUPER^.Cycle();
axesGear(_MasterAxis := MoverArray[MoverToGearTo].AxisRef, _SlaveAxis := THIS^.AxisRef);
moverSequence(ThisMover := THIS^,
				XtsTrack := XtsTrack,
				StateMachine := StateMachine,
				MoverArray := MoverArray);
END_METHOD

METHOD PUBLIC Gear : BOOL
VAR_INPUT
	MasterPosition : MC_LREAL;
	SlavePosition : MC_LREAL;
END_VAR
IF NOT axesGear.Busy THEN
		Gear := axesGear.Sync(MasterPosition := MasterPosition, SlavePosition := SlavePosition);
END_IF
END_METHOD

METHOD inGear : BOOL
VAR_INPUT
END_VAR
inGear := axesGear.gearInCA.InSync;
END_METHOD

METHOD isMaster : BOOL
VAR_INPUT
END_VAR
isMaster := isMasterAxis;
END_METHOD

METHOD masterAxis : UDINT
VAR_INPUT
END_VAR
masterAxis := MoverToGearTo;
END_METHOD

END_FUNCTION_BLOCK

// ---- XTS Class/XtsTrack.TcPOU
FUNCTION_BLOCK XtsTrack EXTENDS PML_Method_Base IMPLEMENTS IXtsTrack 
VAR_INPUT
	TmsSwitch : ITF_TmsSwitch;
END_VAR
VAR_OUTPUT
END_VAR
VAR
	_trackLength : MC_LREAL;
	_homePosition : MC_LREAL;
	HomeSpeed : MC_LREAL := 1000.0;
	mcCollisionGroup : CollisionGroup;
	_XtsTrackHardware : IXtsHardware;
	EnableSequence : XtsEnableSequence(mcCollisionGroup);
	DisableSequence : XtsDisableSequence(mcCollisionGroup);
	GroupStop : StopMoverGroup(mcCollisionGroup);
	State : INT;	
	i : DINT;
	AtHome: BOOL;
	_tracks : UDINT;
	_MoverArray : ARRAY[1..SystemParameters.NumberOfMovers] OF IMover;
END_VAR

METHOD PROTECTED Aborting : BOOL
VAR_INPUT
END_VAR
CASE State OF
	0:
		DisableSequence.Disable();
		State := 1;
			
	1:
		IF DisableSequence.Done THEN
			State := 0;
			ipackml.SetStateComplete();
		END_IF
END_CASE
END_METHOD

METHOD PUBLIC ActivateTracksInMovers : BOOL
VAR_INPUT
END_VAR
VAR
	iTmsMover : ITmsMover;
END_VAR
FOR i := 1 TO SystemParameters.NumberOfMovers DO
	IF __QUERYINTERFACE(_MoverArray[i],iTmsMover) THEN
		iTmsMover.ActivateTrack(newTrack := iTmsMover.ActiveTrack);
	END_IF
END_FOR
ActivateTracksInMovers := true;
END_METHOD

METHOD PROTECTED Clearing : BOOL
VAR_INPUT
END_VAR
CASE State OF
	0:
		IF EnableSequence.Enable() THEN
			State := 1;
		END_IF	
		
	1:
		IF EnableSequence.Done THEN
			State := 2;
		END_IF
		
	2:
		IF ActivateTracksInMovers() THEN
			ipackml.SetStateComplete();
			State := 0;
		END_IF
END_CASE
END_METHOD

METHOD PUBLIC Cycle : BOOL
VAR_INPUT
END_VAR
SUPER^.Cycle();
_XtsTrackHardware.Cycle();
EnableSequence.Cycle();
DisableSequence.Cycle();
GroupStop.Cycle();
mcCollisionGroup.Cycle();
END_METHOD

METHOD PUBLIC GetTMSMoverInterface : BOOL
VAR_INPUT
END_VAR
VAR
	iTmsMover : ITmsMover;
END_VAR
FOR i := 1 TO SystemParameters.NumberOfMovers DO
	IF __QUERYINTERFACE(_MoverArray[i],iTmsMover) THEN
		iTmsMover.SetMoverInterface(MoverInterface := _XtsTrackHardware.GetMoverEnvInterface(DINT_TO_UINT(i)));
	END_IF
END_FOR
END_METHOD

PROPERTY PUBLIC HomePosition : mc_lreal
GET
HomePosition := _homePosition;
END_GET
SET
_homePosition := HomePosition;
END_SET
END_PROPERTY

PROPERTY MoverArray : array[1..SystemParameters.NumberOfMovers] of IMover
GET
MoverArray := _MoverArray;
END_GET
SET
_MoverArray := MoverArray;
EnableSequence.MoverArray := MoverArray;
DisableSequence.MoverArray := MoverArray;
END_SET
END_PROPERTY

METHOD PUBLIC MoverHomeSequence : BOOL
VAR_INPUT
END_VAR
FOR i := 1 TO SystemParameters.NumberOfMovers DO
	_MoverArray[i].MoveTo(Position := _homePosition, Velocity := HomeSpeed, BackwardMove := FALSE);
END_FOR 
MoverHomeSequence := TRUE;
END_METHOD

METHOD PROTECTED Resetting : BOOL
VAR_INPUT
END_VAR
CASE State OF
	0:
		IF MoverHomeSequence() THEN
			State := 1;
		END_IF
	
	1:
		AtHome := TRUE;
		FOR i := 1 TO SystemParameters.NumberOfMovers DO
				AtHome := AtHome AND _MoverArray[i].isStationary();
		END_FOR 
		IF AtHome THEN
			State := 0;
			ipackml.SetStateComplete();	
		END_IF	
END_CASE
END_METHOD

METHOD PROTECTED Stopping : BOOL
VAR_INPUT
END_VAR
CASE State OF
	0:
		GroupStop.Execute();
		State := 1;
		
	1:
		IF GroupStop.Done THEN
			State := 0;
			ipackml.SetStateComplete();
		END_IF
END_CASE
END_METHOD

PROPERTY PUBLIC TrackLength : mc_lreal
GET
TrackLength := _trackLength;
END_GET
SET // PUBLIC
_trackLength := TrackLength;
END_SET
END_PROPERTY

PROPERTY PUBLIC Tracks : UDINT
GET
Tracks := _tracks;
END_GET
SET
_tracks := Tracks;
END_SET
END_PROPERTY

METHOD PROTECTED Undefined : BOOL
VAR_INPUT
END_VAR
IF _XtsTrackHardware.IsHardwareOk() THEN
	GetTMSMoverInterface();
	ipackml.PmlStateCommand(Command := E_PMLCommand.ePMLCommand_Abort);
END_IF
END_METHOD

PROPERTY XtsHardware : IXtsHardware
GET
XtsHardware := _XtsTrackHardware;
END_GET
SET
_XtsTrackHardware := XtsHardware;
END_SET
END_PROPERTY

END_FUNCTION_BLOCK

// ---- PackML_Method_Pattern/PML_Method_Base.TcPOU
FUNCTION_BLOCK PML_Method_Base EXTENDS CyclicBase
VAR_INPUT
END_VAR
VAR_OUTPUT
END_VAR
VAR
	ipackml : IPmlStateMachine;
END_VAR

METHOD PROTECTED Aborted : BOOL
VAR_INPUT
END_VAR
END_METHOD

METHOD PROTECTED Aborting : BOOL
VAR_INPUT
END_VAR
ipackml.SetStateComplete();
END_METHOD

METHOD PROTECTED Clearing : BOOL
VAR_INPUT
END_VAR
ipackml.SetStateComplete();
END_METHOD

METHOD PROTECTED Completed : BOOL
VAR_INPUT
END_VAR
END_METHOD

METHOD PROTECTED Completing : BOOL
VAR_INPUT
END_VAR
ipackml.SetStateComplete();
END_METHOD

METHOD PUBLIC Cycle : BOOL
VAR_INPUT
END_VAR
CASE ipackml.GetCurrentState() OF
	E_PMLState.ePMLState_Clearing:
		Clearing();
	E_PMLState.ePMLState_Aborted:
		Aborted();
	E_PMLState.ePMLState_Aborting:
		Aborting();
	E_PMLState.ePMLState_Complete:
		Completed();
	E_PMLState.ePMLState_Completing:
		Completing();
	E_PMLState.ePMLState_Execute:
		Execute();
	E_PMLState.ePMLState_Held:
		Held();
	E_PMLState.ePMLState_Holding:
		Holding();
	E_PMLState.ePMLState_Idle:
		Idle();
	E_PMLState.ePMLState_Resetting:
		Resetting();
	E_PMLState.ePMLState_Starting:
		Starting();
	E_PMLState.ePMLState_Stopped:
		Stopped();
	E_PMLState.ePMLState_Stopping:
		Stopping();
	E_PMLState.ePMLState_Suspended:
		Suspended();
	E_PMLState.ePMLState_Suspending:
		Suspending();
	E_PMLState.ePMLState_Undefined:
		Undefined();
	E_PMLState.ePMLState_Unholding:
		Unholding();
	E_PMLState.ePMLState_Unsuspending:
		Unsuspending();
END_CASE
END_METHOD

METHOD PROTECTED Execute : BOOL
VAR_INPUT
END_VAR
END_METHOD

METHOD PROTECTED Held : BOOL
VAR_INPUT
END_VAR
END_METHOD

METHOD PROTECTED Holding : BOOL
VAR_INPUT
END_VAR
ipackml.SetStateComplete();
END_METHOD

METHOD PROTECTED Idle : BOOL
VAR_INPUT
END_VAR
END_METHOD

PROPERTY PUBLIC PackMLStateMachine : IPmlStateMachine
GET
PackMLStateMachine := ipackml;
END_GET
SET
ipackml := PackMLStateMachine;
END_SET
END_PROPERTY

METHOD PROTECTED Resetting : BOOL
VAR_INPUT
END_VAR
ipackml.SetStateComplete();
END_METHOD

METHOD PROTECTED Starting : BOOL
VAR_INPUT
END_VAR
ipackml.SetStateComplete();
END_METHOD

METHOD PROTECTED Stopped : BOOL
VAR_INPUT
END_VAR
END_METHOD

METHOD PROTECTED Stopping : BOOL
VAR_INPUT
END_VAR
ipackml.SetStateComplete();
END_METHOD

METHOD PROTECTED Suspended : BOOL
VAR_INPUT
END_VAR
END_METHOD

METHOD PROTECTED Suspending : BOOL
VAR_INPUT
END_VAR
ipackml.SetStateComplete();
END_METHOD

METHOD PROTECTED Undefined : BOOL
VAR_INPUT
END_VAR
END_METHOD

METHOD PROTECTED Unholding : BOOL
VAR_INPUT
END_VAR
ipackml.SetStateComplete();
END_METHOD

METHOD PROTECTED Unsuspending : BOOL
VAR_INPUT
END_VAR
ipackml.SetStateComplete();
END_METHOD

END_FUNCTION_BLOCK

// ---- XTS Class/Xts Collision Group/CollisionGroup.TcPOU
FUNCTION_BLOCK CollisionGroup extends CyclicBase IMPLEMENTS ICollisionGroup
VAR_INPUT
END_VAR
VAR_OUTPUT
END_VAR
VAR
	stGroupInformation : CAGroupInfo;
	_caGroup : Tc3_McCoordinatedMotion.AXES_GROUP_REF;
	readStatus : Tc3_McCoordinatedMotion.MC_GroupReadStatus;
	resetCAGroup : ResetGroup(THIS^);
	enableCAGroup : EnableGroup(THIS^);
	disableCAGroup : DisableGroup(this^);
END_VAR

METHOD Cycle : BOOL
VAR_INPUT
END_VAR
readStatus(
	AxesGroup:= _caGroup, 
	Enable:= TRUE );
resetCAGroup.Cycle();
enableCAGroup.Cycle();
disableCAGroup.Cycle();

//Cyclic get CaGroup information
stGroupInformation.sName := 'MainCAGroup';
stGroupInformation.eGroupState := _caGroup.NcToPlc.Common.GroupStatus.State;
stGroupInformation.nAxesCount	:= UDINT_TO_INT(_caGroup.NcToPlc.Common.GroupAxesCount);
stGroupInformation.nId			:= _caGroup.NcToPlc.Common.GroupOID;
END_METHOD

METHOD Disable : BOOL
VAR_INPUT
END_VAR
IF NOT disableCAGroup.Busy THEN
	disableCAGroup.Execute();
END_IF
END_METHOD

METHOD Enable : BOOL
VAR_INPUT
END_VAR
IF NOT enableCAGroup.Busy THEN
	enableCAGroup.Execute();
END_IF
END_METHOD

PROPERTY GroupRef : reference to AXES_GROUP_REF
GET
GroupRef REF= _caGroup;
END_GET
END_PROPERTY

PROPERTY GroupState : CAGroupStatus
GET
IF readStatus.GroupDisabled THEN
	GroupState := CAGroupStatus.mcGroupStateDisabled;
ELSIF readStatus.GroupErrorStop THEN
	GroupState := CAGroupStatus.mcGroupStateErrorStop;
ELSIF readStatus.GroupHoming THEN
	GroupState := CAGroupStatus.mcGroupStateHoming;
ELSIF readStatus.GroupMoving THEN
	GroupState := CAGroupStatus.mcGroupStateMoving;
ELSIF readStatus.GroupNotReady THEN
	GroupState := CAGroupStatus.mcGroupStateNotReady;
ELSIF readStatus.GroupStandby THEN
	GroupState := CAGroupStatus.mcGroupStateStandby;
ELSIF readStatus.GroupStopping THEN
	GroupState := CAGroupStatus.mcGroupStateStopping;
ELSIF readStatus.Error THEN
	GroupState := CAGroupStatus.mcGroupError;
END_IF
END_GET
END_PROPERTY

METHOD Reset : BOOL
IF NOT resetCAGroup.Busy THEN
	resetCAGroup.Execute();
END_IF
END_METHOD

END_FUNCTION_BLOCK

// ---- Tasks/ResetGroup.TcPOU
{attribute 'hide_all_locals'}
FUNCTION_BLOCK ResetGroup EXTENDS TaskBase
VAR_INPUT
END_VAR
VAR_OUTPUT
END_VAR
VAR
	groupReset			: MC_GroupReset;
	_caGroup			: ICollisionGroup;
	_resetGroup : BOOL;
	Logger : TcMessage_Ext;
END_VAR

METHOD Abort : BOOL
groupReset.Execute := FALSE;
State := 0;
Abort := true;
END_METHOD

METHOD Cycle : BOOL
VAR_INPUT
END_VAR
CASE State OF
	0:
		IF _resetGroup THEN
			_done := FALSE;
			_error := FALSE;
			_busy := TRUE;
			groupReset.Execute := TRUE;
			IF groupReset.Busy THEN
				State := 10;
				_resetGroup := FALSE;
				Logger.Send(TC_EVENTS.XtsCAGroupEvents.CAGroupResetting,'');
			END_IF
		END_IF
	
	10:
		IF NOT groupReset.Busy THEN
			IF groupReset.Done THEN
				_done := TRUE;
				Logger.Send(TC_EVENTS.XtsCAGroupEvents.CAGroupResetDone,'');
			ELSIF groupReset.Error THEN
				_error := TRUE;
				Logger.Send(TC_EVENTS.XtsCAGroupEvents.CAGroupResetError,'');
			END_IF
			_busy := FALSE;
			groupReset.Execute := false;
			State := 0;
		END_IF
END_CASE


groupReset(AxesGroup := _caGroup.GroupRef);
END_METHOD

METHOD Execute : BOOL
Execute := _resetGroup := true;
END_METHOD

METHOD FB_init : BOOL
VAR_INPUT
	bInitRetains : BOOL; // if TRUE, the retain variables are initialized (warm start / cold start)
	bInCopyCode : BOOL;  // if TRUE, the instance afterwards gets moved into the copy code (online change)
	CAGroup : ICollisionGroup;	
END_VAR
_caGroup := CAGroup;
END_METHOD

END_FUNCTION_BLOCK

// ---- Tasks/EnableGroup.TcPOU
{attribute 'hide_all_locals'}
FUNCTION_BLOCK EnableGroup EXTENDS TaskBase
VAR_INPUT
END_VAR
VAR_OUTPUT
END_VAR
VAR
	groupEnable			: MC_GroupEnable;
	_caGroup			: ICollisionGroup;
	_enableGroup : BOOL;
	Logger : TcMessage_Ext;
END_VAR

METHOD Abort : BOOL
groupEnable.Execute := FALSE;
Abort := TRUE;
State := 0;
END_METHOD

METHOD Cycle : BOOL
VAR_INPUT
END_VAR
CASE State OF
	0:
		IF _enableGroup THEN
			_done := FALSE;
			_error := FALSE;
			_busy := TRUE;
			groupEnable.Execute := TRUE;
			IF groupEnable.Busy THEN
				State := 10;
				_enableGroup := FALSE;
				logger.Send(TC_EVENTS.XtsCAGroupEvents.CAGroupEnabling,'');
			END_IF
		END_IF
	
	10:
		IF NOT groupEnable.Busy THEN
			IF groupEnable.Done THEN
				_done := TRUE;
				logger.Send(TC_EVENTS.XtsCAGroupEvents.CAGroupEnabled,'');
			ELSIF groupEnable.Error THEN
				_error := TRUE;
				logger.Send(TC_EVENTS.XtsCAGroupEvents.CAGroupEnableError,'');
			END_IF
			_busy := FALSE;
			groupEnable.Execute := false;
			State := 0;
		END_IF
END_CASE


groupEnable(AxesGroup := _caGroup.GroupRef);
END_METHOD

METHOD Execute : BOOL
Execute := _enableGroup := true;
END_METHOD

METHOD FB_init : BOOL
VAR_INPUT
	bInitRetains : BOOL; // if TRUE, the retain variables are initialized (warm start / cold start)
	bInCopyCode : BOOL;  // if TRUE, the instance afterwards gets moved into the copy code (online change)
	CAGroup : ICollisionGroup;	
END_VAR
_caGroup := CAGroup;
END_METHOD

END_FUNCTION_BLOCK

// ---- Tasks/DisableGroup.TcPOU
{attribute 'hide_all_locals'}
FUNCTION_BLOCK DisableGroup EXTENDS TaskBase
VAR_INPUT
END_VAR
VAR_OUTPUT
END_VAR
VAR
	groupDisable			: MC_GroupDisable;
	_caGroup			: ICollisionGroup;
	_disableGroup : BOOL;
	Logger : TcMessage_Ext;
END_VAR

METHOD Abort : BOOL
State := 0;
groupDisable.Execute := FALSE;
Abort := true;
END_METHOD

METHOD Cycle : BOOL
VAR_INPUT
END_VAR
CASE State OF
	0:
		IF _disableGroup THEN
			_done := FALSE;
			_error := FALSE;
			_busy := TRUE;
			groupDisable.Execute := TRUE;
			IF groupDisable.Busy THEN
				_disableGroup := FALSE;
				State := 10;
				logger.Send(TC_EVENTS.XtsCAGroupEvents.CAGroupDisabling,'');
			END_IF
		END_IF
	
	10:
		IF NOT groupDisable.Busy THEN
			IF groupDisable.Done THEN
				_done := TRUE;
				logger.Send(TC_EVENTS.XtsCAGroupEvents.CAGroupDisabled,'');
			ELSIF groupDisable.Error THEN
				_error := TRUE;
				logger.Send(TC_EVENTS.XtsCAGroupEvents.CAGroupDisableError,'');
			END_IF
			_busy := FALSE;
			groupDisable.Execute := false;
			State := 0;
		END_IF
END_CASE


groupDisable(AxesGroup := _caGroup.GroupRef);
END_METHOD

METHOD Execute : BOOL
Execute := _disableGroup := TRUE;
END_METHOD

METHOD FB_init : BOOL
VAR_INPUT
	bInitRetains : BOOL; // if TRUE, the retain variables are initialized (warm start / cold start)
	bInCopyCode : BOOL;  // if TRUE, the instance afterwards gets moved into the copy code (online change)
	CAGroup : ICollisionGroup;
END_VAR
_caGroup := CAGroup;
END_METHOD

END_FUNCTION_BLOCK

// ---- Tasks/XtsEnableSequence.TcPOU
FUNCTION_BLOCK XtsEnableSequence EXTENDS TaskBase
VAR_INPUT
END_VAR
VAR_OUTPUT
END_VAR
VAR
	_collisionGroup : ICollisionGroup;
	addMover : AddMoverToGroupTask(_collisionGroup);
	moverNumbers : DINT;
	AllMoversEnabled: BOOL;
	EnableTrigger : BOOL;	
	Logger : TcMessage_Ext;
	arrMovers : ARRAY[1..SystemParameters.NumberOfMovers] OF IMover;
END_VAR

METHOD Abort : BOOL
EnableTrigger := FALSE;
State := 0;
addMover.Abort();
END_METHOD

PROPERTY Busy : BOOL
GET
Busy := _busy;
END_GET
END_PROPERTY

METHOD Cycle : BOOL
VAR_INPUT
END_VAR
CASE State OF
	0:
		IF EnableTrigger THEN
			State := 10;
			EnableTrigger := FALSE;
			moverNumbers := 1;
			_busy := TRUE;
			_done := FALSE;
			_Error := FALSE;
		END_IF
		
	10:
		FOR moverNumbers := 1 TO SystemParameters.NumberOfMovers DO
			arrMovers[moverNumbers].ResetAxis();
		END_FOR
		moverNumbers := 1;
		State := 20;
		
	20:
		IF _collisionGroup.GroupState = CAGroupStatus.mcGroupStateErrorStop THEN
			_collisionGroup.Reset();
			Logger.Send(TC_EVENTS.XtsCAGroupEvents.CAGroupReset,'');
		END_IF
		State := 30;
		
	30:
		arrMovers[moverNumbers].IdentInGroup := DINT_TO_INT( moverNumbers);
		addMover.AddMover(MoverToAdd := arrMovers[moverNumbers]);
		logger.Send(TC_EVENTS.XtsCAGroupEvents.AddingMoverToGroup,DINT_TO_STRING(moverNumbers));
		State := 40;
		
	40:
		IF addMover.Done THEN
			IF moverNumbers <> SystemParameters.NumberOfMovers THEN
				moverNumbers := moverNumbers + 1;
				State := 30;
			ELSE
				logger.Send(TC_EVENTS.XtsCAGroupEvents.AllMoversAdded,'');
				FOR moverNumbers := 1 TO SystemParameters.NumberOfMovers DO
					arrMovers[moverNumbers].EnableAxis();
				END_FOR
				State := 50;
			END_IF
		END_IF
		
	50:
		AllMoversEnabled := TRUE;
		FOR moverNumbers := 1 TO SystemParameters.NumberOfMovers DO
			AllMoversEnabled := TRUE AND arrMovers[moverNumbers].isEnabled();
		END_FOR
		IF AllMoversEnabled THEN
			logger.Send(TC_EVENTS.XtsCAGroupEvents.AllMoversEnabled,'');
			_collisionGroup.Enable();
			logger.Send(TC_EVENTS.XtsCAGroupEvents.CAGroupEnable,'');
			State := 60;
		END_IF
		
	60:
		IF _collisionGroup.GroupState = 2 THEN
			State := 0;
			_busy := FALSE;
			_done := true;
		END_IF
END_CASE

addMover.Cycle();
END_METHOD

PROPERTY Done : BOOL
GET
Done := _done;
END_GET
END_PROPERTY

METHOD Enable : BOOL
VAR_INPUT
END_VAR
IF NOT _busy THEN
	EnableTrigger := Enable := true;
END_IF
END_METHOD

PROPERTY Error : BOOL
GET
Error := _Error;
END_GET
END_PROPERTY

METHOD FB_init : BOOL
VAR_INPUT
	bInitRetains : BOOL; // if TRUE, the retain variables are initialized (warm start / cold start)
	bInCopyCode : BOOL;  // if TRUE, the instance afterwards gets moved into the copy code (online change)
	collisionGroup : ICollisionGroup;
END_VAR
_collisionGroup := collisionGroup;
addMover.FB_init(FALSE, FALSE, collisionGroup);
END_METHOD

PROPERTY MoverArray : array[1..SystemParameters.NumberOfMovers] of IMover
GET
MoverArray := arrMovers;
END_GET
SET
arrMovers := MoverArray;
END_SET
END_PROPERTY

END_FUNCTION_BLOCK

// ---- Tasks/AddMoverToGroupTask.TcPOU
FUNCTION_BLOCK AddMoverToGroupTask EXTENDS TaskBase
VAR_INPUT
END_VAR
VAR_OUTPUT
END_VAR
VAR
	AddtoGrp			: MC_AddAxisToGroup;
	_caGroup			: ICollisionGroup;
	_axis				: reference TO AXIS_REF;
	_addMover : BOOL;
	_moverNumber : UDINT;
END_VAR

METHOD Abort : BOOL
AddtoGrp.Execute := FALSE;
Abort := true;
State := 0;
END_METHOD

METHOD AddMover : BOOL
VAR_INPUT
	MoverToAdd : IMover;
END_VAR
_axis REF= MoverToAdd.AxisRef;
_moverNumber := INT_TO_UDINT(MoverToAdd.IdentInGroup);
_busy := TRUE;
AddMover := _addMover := TRUE;
END_METHOD

METHOD Cycle : BOOL
VAR_INPUT
END_VAR
CASE State OF
	0:
		IF _addMover THEN
			_done := FALSE;
			_error := FALSE;
			_busy := true;
			AddtoGrp.Execute := TRUE;
			IF AddtoGrp.Busy THEN
				State := 10;
				_addMover := FALSE;
			END_IF
		END_IF
	
	10:
		IF NOT AddtoGrp.Busy THEN
			IF AddtoGrp.Done THEN
				_done := TRUE;
			ELSIF AddtoGrp.Error THEN
				_error := TRUE;
			END_IF
			_busy := FALSE;
			AddtoGrp.Execute := false;
			State := 0;
		END_IF
END_CASE

AddtoGrp(AxesGroup := _caGroup.GroupRef,
			Axis := _axis,
			IdentInGroup := UDINT_TO_IDENTINGROUP(_moverNumber));
END_METHOD

METHOD FB_init : BOOL
VAR_INPUT
	bInitRetains : BOOL; // if TRUE, the retain variables are initialized (warm start / cold start)
	bInCopyCode : BOOL;  // if TRUE, the instance afterwards gets moved into the copy code (online change)
	collisionGroup : ICollisionGroup;	
END_VAR
_caGroup := collisionGroup;
END_METHOD

END_FUNCTION_BLOCK

// ---- Tasks/XtsDisableSequence.TcPOU
FUNCTION_BLOCK XtsDisableSequence EXTENDS TaskBase
VAR_INPUT
END_VAR
VAR_OUTPUT
END_VAR
VAR
	_collisionGroup : ICollisionGroup;
	removeAllAxes : RemoveAllMoverFromGroup(_collisionGroup);
	grpStop : StopMoverGroup(_collisionGroup);
	DisableTrigger: BOOL;
	moverNumbers : DINT := 1;
	AllMoversDisabled: BOOL;	
	Logger : TcMessage_Ext;
	arrMovers : ARRAY[1..SystemParameters.NumberOfMovers] OF IMover;
END_VAR

METHOD Abort : BOOL
DisableTrigger := FALSE;
State := 0;
removeAllAxes.Abort();
grpStop.Abort();
END_METHOD

PROPERTY Busy : BOOL
GET
Busy := _busy;
END_GET
END_PROPERTY

METHOD Cycle : BOOL
VAR_INPUT
END_VAR
CASE State OF
	0:
		IF DisableTrigger THEN
			DisableTrigger := FALSE;
			_busy := TRUE;
			_done := FALSE;
			_Error := FALSE;
			IF _collisionGroup.GroupState = CAGroupStatus.mcGroupStateMoving THEN
				Logger.Send(TC_EVENTS.XtsCAGroupEvents.CAGroupStop,'');
				grpStop.Execute();
				State := 10;
			ELSE
				State := 20;
				removeAllAxes.RemoveAllMover();
				Logger.Send(TC_EVENTS.XtsCAGroupEvents.CaGroupRemoveMovers,'');
			END_IF
		END_IF
		
	10:
		IF grpStop.Done THEN
			State := 20;
			Logger.Send(TC_EVENTS.XtsCAGroupEvents.CaGroupRemoveMovers,'');
			removeAllAxes.RemoveAllMover();
		END_IF
	
	20:
		IF removeAllAxes.Done THEN
			FOR moverNumbers := 1 TO SystemParameters.NumberOfMovers DO
				arrMovers[moverNumbers].IdentInGroup := 0;
				arrMovers[moverNumbers].DisableAxis();
			END_FOR
			State := 30;
		END_IF
		
	30:
		AllMoversDisabled := TRUE;
		FOR moverNumbers := 1 TO SystemParameters.NumberOfMovers DO
			AllMoversDisabled := TRUE AND NOT arrMovers[moverNumbers].isEnabled();
		END_FOR
		IF AllMoversDisabled THEN
			logger.Send(TC_EVENTS.XtsCAGroupEvents.AllMoversDisabled,'');
			State := 40;
			_collisionGroup.Disable();
			logger.Send(TC_EVENTS.XtsCAGroupEvents.CAGroupDisable,'');
		END_IF
	40:
		IF _collisionGroup.GroupState = CAGroupStatus.mcGroupStateErrorStop THEN
			_collisionGroup.Reset();
			Logger.Send(TC_EVENTS.XtsCAGroupEvents.CAGroupReset,'');
		END_IF	
		State := 50;
		
	50:
		IF _collisionGroup.GroupState = 1 THEN
			State := 0;
			grpStop.Deceleration := Tc3_Mc3Definitions.MC_DEFAULT;
			grpStop.Jerk := Tc3_Mc3Definitions.MC_DEFAULT;
			
			_busy := FALSE;
			_done := true;
		END_IF
END_CASE

removeAllAxes.Cycle();
grpStop.Cycle();
END_METHOD

METHOD Disable : BOOL
VAR_INPUT
END_VAR
DisableTrigger := true;
END_METHOD

PROPERTY Done : BOOL
GET
Done := _done;
END_GET
END_PROPERTY

PROPERTY Error : BOOL
GET
Error := _Error;
END_GET
END_PROPERTY

METHOD FB_init : BOOL
VAR_INPUT
	bInitRetains : BOOL; // if TRUE, the retain variables are initialized (warm start / cold start)
	bInCopyCode : BOOL;  // if TRUE, the instance afterwards gets moved into the copy code (online change)
	collisionGroup : ICollisionGroup;
END_VAR
_collisionGroup := collisionGroup;
removeAllAxes.FB_init(FALSE, FALSE, CAGroup := collisionGroup);
grpStop.FB_init(FALSE,FALSE,CAGroup := collisionGroup);
END_METHOD

PROPERTY MoverArray : array[1..SystemParameters.NumberOfMovers] of IMover
GET
MoverArray := arrMovers;
END_GET
SET
arrMovers := MoverArray;
END_SET
END_PROPERTY

METHOD SetEmergencyDynamics : BOOL
VAR_INPUT
END_VAR
grpStop.Deceleration := Tc3_Mc3Definitions.MC_MAXIMUM;
grpStop.Jerk := Tc3_Mc3Definitions.MC_MAXIMUM;
END_METHOD

END_FUNCTION_BLOCK

// ---- Tasks/RemoveAllMoverFromGroup.TcPOU
FUNCTION_BLOCK RemoveAllMoverFromGroup EXTENDS TaskBase
VAR_INPUT
END_VAR
VAR_OUTPUT
END_VAR
VAR
	RemoveAllFromGrp			: MC_UngroupAllAxes;
	_caGroup			: ICollisionGroup;
	_removeAllMovers : BOOL;
	_errorId: UDINT;
	Logger : TcMessage_Ext;
END_VAR

METHOD Abort : BOOL
RemoveAllFromGrp.Execute := FALSE;
Abort := true;
State := 0;
END_METHOD

METHOD Cycle : BOOL
VAR_INPUT
END_VAR
CASE State OF
	0:
		IF _removeAllMovers THEN
			_done := FALSE;
			_error := FALSE;
			_busy := TRUE;
			RemoveAllFromGrp.Execute := TRUE;
			IF RemoveAllFromGrp.Busy THEN
				_removeAllMovers := FALSE;
				State := 10;
				logger.Send(TC_EVENTS.XtsCAGroupEvents.CAGroupRemoving,'');
			END_IF
		END_IF
		
	10:
		IF NOT RemoveAllFromGrp.Busy THEN
			IF RemoveAllFromGrp.Done THEN
				_done := TRUE;
				logger.Send(TC_EVENTS.XtsCAGroupEvents.AllMoversRemoved,'');
			ELSIF RemoveAllFromGrp.Error THEN
				_error := TRUE;
				_errorId := RemoveAllFromGrp.ErrorId;
				Logger.Send(TC_EVENTS.XtsCAGroupEvents.CAGroupRemoveError,'');
			END_IF
			_busy := FALSE;
			RemoveAllFromGrp.Execute := false;
			State := 0;
		END_IF
END_CASE


RemoveAllFromGrp(AxesGroup := _caGroup.GroupRef);
END_METHOD

METHOD FB_init : BOOL
VAR_INPUT
	bInitRetains : BOOL; // if TRUE, the retain variables are initialized (warm start / cold start)
	bInCopyCode : BOOL;  // if TRUE, the instance afterwards gets moved into the copy code (online change)
	CAGroup : ICollisionGroup;	
END_VAR
_caGroup := CAGroup;
END_METHOD

METHOD RemoveAllMover : BOOL
RemoveAllMover := _removeAllMovers := true;
END_METHOD

END_FUNCTION_BLOCK

// ---- Tasks/StopMoverGroup.TcPOU
FUNCTION_BLOCK StopMoverGroup EXTENDS TaskBase
VAR_INPUT
END_VAR
VAR_OUTPUT
END_VAR
VAR
	groupStop			: MC_GroupStop;
	_caGroup			: ICollisionGroup;
	_stopGroup : BOOL;
	_jerk : MC_LREAL;
	_deceleration : MC_LREAL;
	Logger : TcMessage_Ext;
END_VAR

METHOD Abort : BOOL
groupStop.Execute := FALSE;
State := 0;
Abort := true;
END_METHOD

METHOD Cycle : BOOL
VAR_INPUT
END_VAR
CASE State OF
	0:
		IF _stopGroup THEN
			_done := FALSE;
			_error := FALSE;
			_busy := TRUE;
			groupStop.Execute := TRUE;
			IF groupStop.Busy THEN
				State := 10;
				_stopGroup := FALSE;
				Logger.Send(TC_EVENTS.XtsCAGroupEvents.CAGroupStopping,'');
			END_IF
		END_IF
	10:
		IF groupStop.Done THEN
			_done := TRUE;
			Logger.Send(TC_EVENTS.XtsCAGroupEvents.CAGroupStopped,'');
		ELSIF groupStop.Error THEN
			_error := TRUE;
			Logger.Send(TC_EVENTS.XtsCAGroupEvents.CAGroupStopError,'');
		END_IF
		IF _done OR _error THEN
			_busy := FALSE;
			groupStop.Execute := FALSE;
			State := 0;
		END_IF
END_CASE


groupStop(AxesGroup := _caGroup.GroupRef);
END_METHOD

PROPERTY PUBLIC Deceleration : MC_LREAL
GET
Deceleration := _deceleration;
END_GET
SET
_deceleration := Deceleration;
END_SET
END_PROPERTY

METHOD Execute : BOOL
_stopGroup := Execute := true;
END_METHOD

METHOD FB_init : BOOL
VAR_INPUT
	bInitRetains : BOOL; // if TRUE, the retain variables are initialized (warm start / cold start)
	bInCopyCode : BOOL;  // if TRUE, the instance afterwards gets moved into the copy code (online change)
	CAGroup : ICollisionGroup;
END_VAR
_caGroup := CAGroup;
END_METHOD

PROPERTY PUBLIC Jerk : MC_LREAL
GET
Jerk := _jerk;
END_GET
SET
_jerk := Jerk;
END_SET
END_PROPERTY

END_FUNCTION_BLOCK

// ---- XTS Class/Xts Hardware/XtsHardware.TcPOU
FUNCTION_BLOCK XtsHardware
VAR_INPUT
	Tracks : UDINT;
	TmsSwitch : ITF_TmsSwitch;
END_VAR
VAR_OUTPUT
	XtsHardwareOK : BOOL;
	Xts48VStanding : BOOL;
	Xts24VStanding : BOOL;
END_VAR
VAR
	XtsIoEnvironment : Tc3_XTS_Utility.FB_TcIoXtsEnvironment;
	bInit: BOOL;
	bMoverIdDetectionError		: BOOL;
	bMoverIdDetectionActive		: BOOL;
	bMoverIdDetected : BOOL;
	bTriggerStarted: BOOL;
	f24V: ARRAY[1..SystemParameters.nModuleNumber] OF UINT;
	f48V: ARRAY[1..SystemParameters.nModuleNumber] OF UINT;
	CurrentLive : ARRAY[1..SystemParameters.nModuleNumber] OF DINT;
	MaxCurrent : ARRAY [1..SystemParameters.nModuleNumber] OF DINT;
	nModuleCounter : UINT := 1;
	i: UDINT;
	State : XtsHardwareState;
	Logger : TcMessage_Ext;
	DetectedParts: UDINT;
	DetectedTracks : UDINT;
	DetectedModules : ARRAY[1..10] OF UDINT;
	PartIndex: UINT := 1;
	ModuleIndex : INT := 1;
	XtsHWInfo : XtsHardwareInfo;
END_VAR

IF NOT bInit THEN
	IF XtsIoEnvironment.Init(TRUE) THEN
		XtsIoEnvironment.Init(FALSE);
		bInit := TRUE;
	END_IF
	RETURN;
END_IF

CASE State OF
	XtsHardwareState.Init:
		IF GetTrackAssembly() THEN
			State := XtsHardwareState.SetDetection;
		END_IF
	
	XtsHardwareState.SetDetection:
		IF SetTracksForDetection() THEN
			State := XtsHardwareState.Redetect;
		END_IF
		
	XtsHardwareState.Redetect:
		IF TriggerMoverDetection() THEN
			State := XtsHardwareState.MoversValid;
		END_IF
		
	XtsHardwareState.MoversValid:
		IF getAllMoversValid() THEN
			State := XtsHardwareState.AllMoversFound;
		END_IF
	
	XtsHardwareState.AllMoversFound:
		IF getMoversDetected() THEN
			State := XtsHardwareState.MoverIdDetection;
		END_IF
		
	XtsHardwareState.MoverIdDetection:
		IF TriggerMoverID() THEN
			State := XtsHardwareState.XtsMode;
		END_IF
	
	XtsHardwareState.XtsMode:
		IF IsInSim() THEN
			State := XtsHardwareState.HWReady;
		ELSE
			State := XtsHardwareState.CheckModuleVoltages;
		END_IF
		
	XtsHardwareState.CheckModuleVoltages:
		Xts48VStanding := TRUE;
		Xts24VStanding := TRUE;
		FOR i := 1 TO SystemParameters.nModuleNumber DO
			IF f48V[i] < 46000 THEN
				Xts48VStanding := FALSE;
			END_IF
			IF f24V[i] < 20400 THEN
				Xts24VStanding := FALSE;
			END_IF
		END_FOR
		IF Xts24VStanding AND Xts48VStanding THEN
			State := XtsHardwareState.HWReady;
		END_IF
	
	XtsHardwareState.HWReady:
		XtsHardwareOK := TRUE;
END_CASE

getModuleInfoData();

//CYCLIC update of info
XtsHWInfo.HWState := State;

METHOD getAllMoversValid : BOOL
VAR_INPUT
END_VAR
 IF XtsIoEnvironment.XpuTcIo(1).GetAreAllPositionsValid() THEN
	 getAllMoversValid := TRUE;
	 Logger.Send(TC_EVENTS.XtsHardwareEvents.AllMoversValid,'');
 END_IF
END_METHOD

METHOD getModuleInfoData : BOOL
VAR_INPUT
END_VAR
IF XtsIoEnvironment.XpuTcIo(1).PartTcIo(PartIndex).ModuleCoE(nModuleCounter).InfoData.Update() THEN
	CurrentLive[ModuleIndex]:=XtsIoEnvironment.XpuTcIo(1).PartTcIo(PartIndex).ModuleCoE(nModuleCounter).InfoData.OverallCurrent;
	MaxCurrent[ModuleIndex]:=XtsIoEnvironment.XpuTcIo(1).PartTcIo(PartIndex).ModuleCoE(nModuleCounter).InfoData.MaxOverallCurrentLast500ms;
	f24V[ModuleIndex]:=XtsIoEnvironment.XpuTcIo(1).PartTcIo(PartIndex).ModuleCoE(nModuleCounter).InfoData.AuxiliaryVoltage24V;
	f48V[ModuleIndex]:=XtsIoEnvironment.XpuTcIo(1).PartTcIo(PartIndex).ModuleCoE(nModuleCounter).InfoData.DcLinkVoltage;
	ModuleIndex := ModuleIndex + 1;
	IF nModuleCounter = DetectedModules[PartIndex] THEN
		nModuleCounter := 1;
		IF PartIndex = DetectedParts THEN
			PartIndex := 1;
			ModuleIndex := 1;
		ELSE
			PartIndex := PartIndex + 1;
		END_IF
	ELSE
		nModuleCounter := nModuleCounter + 1;
	END_IF
END_IF
END_METHOD

METHOD PUBLIC GetMoverEnvInterface : I_TcIoXtsXpuMover
VAR_INPUT
	MoverNumber : UINT;
END_VAR
GetMoverEnvInterface := XtsIoEnvironment.XpuTcIo(1).MoverTcIo(MoverNumber);
END_METHOD

METHOD getMoversDetected : BOOL
VAR_INPUT
END_VAR
IF XtsIoEnvironment.XpuTcIo(1).GetDetectedMoverCount() = XtsIoEnvironment.XpuTcIo(1).GetExpectedMoverCount() THEN
	getMoversDetected := TRUE;
	Logger.Send(TC_EVENTS.XtsHardwareEvents.ExpectedMoversDetected,UDINT_TO_STRING(XtsIoEnvironment.XpuTcIo(1).GetExpectedMoverCount()));
ELSE
	getMoversDetected := FALSE;
	Logger.Send(TC_EVENTS.XtsHardwareEvents.ExpectedMoversNotFound,'');
END_IF
END_METHOD

METHOD PUBLIC GetTrackAssembly : BOOL
VAR_INPUT
END_VAR
DetectedTracks :=  XtsIoEnvironment.XpuTcIo(1).GetTrackCount();
IF DetectedTracks <> Tracks THEN
	Logger.Send(TC_EVENTS.XtsHardwareEvents.XtsTracksCountError,'');
	RETURN; 
END_IF
DetectedParts := XtsIoEnvironment.XpuTcIo(1).GetPartCount();
FOR i := 1 TO UDINT_TO_UINT(DetectedParts) DO
	DetectedModules[i] := XtsIoEnvironment.XpuTcIo(1).PartTcIo(UDINT_TO_UINT(i)).GetModuleCount();
END_FOR
GetTrackAssembly := TRUE;

XtsHWInfo.NoOfModules := DetectedModules;
XtsHWInfo.NoOfParts := DetectedParts;
XtsHWInfo.NoOfTracks := DetectedTracks;
END_METHOD

METHOD IsInSim : BOOL
VAR_INPUT
END_VAR
IF  XtsIoEnvironment.XpuTcIo(1).GetOperationMode() = OperationMode.Simulation THEN
	IsInSim := TRUE;
	Logger.Send(TC_EVENTS.XtsHardwareEvents.XtsInSimulationMode,'');
ELSE
	IsInSim := FALSE;
END_IF
END_METHOD

METHOD SetTracksForDetection : BOOL
VAR_INPUT
END_VAR
FOR i:=1 TO XtsIoEnvironment.XpuTcIo(1).GetTrackCount() DO
	XtsIoEnvironment.XpuTcIo(1).TrackTcIo(UDINT_TO_UINT(i)).SetIsIncludedInDetection(FALSE);
END_FOR

IF XtsIoEnvironment.XpuTcIo(1).GetTrackCount() = 1 THEN
	XtsIoEnvironment.XpuTcIo(1).TrackTcIo(1).SetIsIncludedInDetection(TRUE);
	Logger.Send(TC_EVENTS.XtsHardwareEvents.ActiveTracksAddedForDetection, UDINT_TO_STRING(XtsIoEnvironment.XpuTcIo(1).GetTrackCount()));
	SetTracksForDetection := TRUE;
ELSE
	CASE TmsSwitch.Switch OF
		TmsSwitchPosition.Up: 
			XtsIoEnvironment.XpuTcIo(1).TrackTcIo(3).SetIsIncludedInDetection(TRUE);
		TmsSwitchPosition.Middle:
			XtsIoEnvironment.XpuTcIo(1).TrackTcIo(1).SetIsIncludedInDetection(TRUE);
			XtsIoEnvironment.XpuTcIo(1).TrackTcIo(2).SetIsIncludedInDetection(TRUE);
		TmsSwitchPosition.Down:
			;
	END_CASE
	Logger.Send(TC_EVENTS.XtsHardwareEvents.ActiveTracksAddedForDetection, UDINT_TO_STRING(XtsIoEnvironment.XpuTcIo(1).GetTrackCount()));
	SetTracksForDetection := TRUE;
END_IF
END_METHOD

METHOD TriggerMoverDetection : BOOL
VAR_INPUT
END_VAR
XtsIoEnvironment.XpuTcIo(1).TriggerRedetection();
Logger.Send(TC_EVENTS.XtsHardwareEvents.MoverDetectionInitiated,'');
TriggerMoverDetection := true;
END_METHOD

METHOD TriggerMoverID : BOOL
VAR_INPUT
END_VAR
VAR
	
END_VAR
// Mover1 Functionality		
// Check if "MoverIdDetectionMode" has been activated under the XtsProcessingUnit object.
IF XtsIoEnvironment.XpuTcIo(1).GetMoverIdDetectionMode() = E_MoverIdDetectionMode.Mover1
	OR XtsIoEnvironment.XpuTcIo(1).GetMoverIdDetectionMode() = 2 THEN

	// Check if the "MoverIdDetection" has already been started or the Mover1 was found.
	IF NOT (bMoverIdDetectionActive OR bMoverIdDetected OR bTriggerStarted) THEN
		// Trigger the "MoverIdDetection".
		XtsIoEnvironment.XpuTcIo(1).TriggerMoverIdDetection();
		Logger.Send(TC_EVENTS.XtsHardwareEvents.Mover1DetectionStarted,'');
		bTriggerStarted := TRUE;
	END_IF

	// Check for error or success of "MoverIdDetection".
	bMoverIdDetectionError 	:= XtsIoEnvironment.XpuTcIo(1).GetHasMoverIdDetectionError();
	bMoverIdDetected 	:= XtsIoEnvironment.XpuTcIo(1).GetIsMoverIdDetectionValid();
	bMoverIdDetectionActive	:= XtsIoEnvironment.XpuTcIo(1).GetIsMoverIdDetectionActive();
	
	// If the detection has an error, check for errors in output and try again.
	IF bMoverIdDetectionError THEN
		Logger.Send(TC_EVENTS.XtsHardwareEvents.Mover1DetectionFailed,'');
		RETURN; 
	END_IF

	// Do not process any further until the "MoverId" was deteced.
	IF NOT bMoverIdDetected THEN
		RETURN;
	END_IF	
	TriggerMoverID := TRUE;	
	Logger.Send(TC_EVENTS.XtsHardwareEvents.Mover1DetectionComplete,'');
ELSE
	TriggerMoverID := TRUE;
	Logger.Send(TC_EVENTS.XtsHardwareEvents.StandardMoverNumberingComplete,'');
END_IF
END_METHOD

END_FUNCTION_BLOCK

// ---- Tasks/GearInCA.TcPOU
FUNCTION_BLOCK PUBLIC GearInCA IMPLEMENTS ITask
VAR_INPUT
END_VAR
VAR_OUTPUT
END_VAR
VAR
	gearInCA : Tc3_McCollisionAvoidance.MC_GearInPosCA;
	_syncStrategy : Tc3_Mc3Definitions.MC_SYNC_STRATEGY := Tc3_Mc3Definitions.MC_SYNC_STRATEGY.mcSyncStrategyEarly;
	_GearMover: BOOL;
	State : INT;
	_busy : BOOL;
	_done : BOOL;
	_Error : BOOL;
END_VAR
VAR_IN_OUT
	_MasterAxis : Tc2_MC2.AXIS_REF;
	_SlaveAxis : Tc2_MC2.AXIS_REF;
END_VAR

CASE State OF
	0:
		IF _GearMover THEN
			_done := FALSE;
			_error := FALSE;
			_busy := TRUE;
			gearInCA.Execute := TRUE;
			IF gearInCA.Busy THEN
				State := 10;
				_GearMover := FALSE;
			END_IF
		END_IF
		
	10:
		IF gearInCA.InSync THEN
			gearInCA.Execute := FALSE;
			_busy := FALSE;
			_done := TRUE;
			State := 0;
		END_IF
	
END_CASE

IF __ISVALIDREF(_MasterAxis) AND __ISVALIDREF(_SlaveAxis) THEN
	gearInCA(Master := _MasterAxis, Slave := _SlaveAxis, SyncStrategy := _syncStrategy, Velocity := 2000.0, RatioNumerator := 1, Gap := 60.0);
END_IF

METHOD Abort : BOOL
gearInCA.Execute := FALSE;
_GearMover := FALSE;
_busy := false;
Abort := true;
State := 0;
END_METHOD

PROPERTY Busy : BOOL
GET
Busy := _busy;
END_GET
END_PROPERTY

PROPERTY Done : BOOL
GET
Done := _done;
END_GET
END_PROPERTY

PROPERTY Error : BOOL
GET
Error := _Error;
END_GET
END_PROPERTY

METHOD PUBLIC Sync : BOOL
VAR_INPUT
	MasterPosition : MC_LREAL;
	SlavePosition : MC_LREAL;
END_VAR
gearInCA.MasterSyncPosition := MasterPosition;
gearInCA.SlaveSyncPosition := SlavePosition;
_GearMover := true;
END_METHOD

PROPERTY PUBLIC SyncStrategy : mc_sync_strategy
GET
SyncStrategy := _syncStrategy;
END_GET
SET
_syncStrategy := SyncStrategy;
END_SET
END_PROPERTY

END_FUNCTION_BLOCK

// ---- Mover Class/TMS_Mover.TcPOU
FUNCTION_BLOCK TMS_Mover EXTENDS FB_Mover IMPLEMENTS ITmsMover
VAR
	ActivateATrack : ActivateTrackForMover(_axis);
	mcReadTrackPositions : Tc3_McCollisionAvoidance.MC_ReadTrackPositions;
	axesMoveModuloTo 		: MoveModuloMoverToPosition(_axis) := (Gap := 100.0);
	_stOptions : ST_MoveAbsoluteCAOptions;
	ipTcIoXtsMover			: I_TcIoXtsXpuMover;
	stTmsActPositions			: ST_PositionInfo;
END_VAR

METHOD ActivateTrack : BOOL
VAR_INPUT
	newTrack : OTCID;
END_VAR
IF NOT ActivateATrack.Busy THEN
	ActivateATrack.Execute(Track := newTrack);
	ActivateTrack := TRUE;
END_IF
END_METHOD

PROPERTY ActiveTrack : OTCID
GET
ActiveTrack := stTmsActPositions.nTrackObjectid;
END_GET
END_PROPERTY

METHOD PUBLIC  Cycle : BOOL
VAR_INPUT
END_VAR
SUPER^.Cycle();
IF _identInGroup <> 0 THEN
	mcReadTrackPositions(
		Axis:= THIS^._axis, 
		Enable:= TRUE, 
		Valid=> , 
		Busy=> , 
		TrackPosition=> , 
		TrackId=> , 
		PartPosition=> , 
		PartId=> , 
		Error=> , 
		ErrorId=> );
END_IF
ActivateATrack.Cycle();
IF ActivateATrack.Done THEN 
	_stOptions.PositionReferenceSystem :=  ActivateATrack.NewTrackId;
	axesMoveModuloTo.Options := _stOptions;
END_IF

IF ipTcIoXtsMover <> 0 THEN
	stTmsActPositions:=ipTcIoXtsMover.GetPositionInfo();
END_IF

axesMoveModuloTo.Cycle();
END_METHOD

METHOD PUBLIC HasCommand : BOOL
VAR_INPUT
END_VAR
HasCommand := axesMoveModuloTo.Busy;
END_METHOD

METHOD isAtPosition : BOOL
VAR_INPUT
	position : MC_LREAL;
END_VAR

VAR
	moduloPos: DINT;
END_VAR
//Create modulo position 
//moduloPos := LREAL_TO_DINT(stTmsActPositions.fTrackPosition) MOD LREAL_TO_DINT(_trackLength);
IF position > 1 THEN
	IF stTmsActPositions.fTrackPosition < position + 1 AND stTmsActPositions.fTrackPosition > position - 1 THEN
		isAtPosition := TRUE;
	END_IF  
ELSE
	IF stTmsActPositions.fTrackPosition < position + 1 AND stTmsActPositions.fTrackPosition > 0.0  
		OR stTmsActPositions.fTrackPosition < _trackLength AND stTmsActPositions.fTrackPosition > _trackLength - 1 THEN
		isAtPosition := TRUE;
	END_IF
END_IF
END_METHOD

METHOD PUBLIC isPastPosition : BOOL
VAR_INPUT
	position : MC_LREAL;
END_VAR
IF position > 1 THEN
	IF stTmsActPositions.fTrackPosition > position THEN
		isPastPosition := TRUE;
	END_IF  
END_IF
END_METHOD

METHOD PUBLIC MoveTo : BOOL
VAR_INPUT
	Position : MC_LREAL;
	Velocity : MC_LREAL;
	BackwardMove : BOOL;
END_VAR
IF NOT THIS^.isAtPosition(position := Position) THEN
	IF NOT axesMoveModuloTo.Busy THEN
		THIS^.axesMoveModuloTo.MoveTo(Position := Position, Velocity := Velocity, Direction := Tc2_MC2.MC_Direction.MC_Positive_Direction, Turns := 0);
		MoveTo := TRUE;
		_targetPos := Position;
	END_IF
END_IF
END_METHOD

METHOD PUBLIC SetMoverInterface : BOOL
VAR_INPUT
	MoverInterface : I_TcIoXtsXpuMover;
END_VAR
ipTcIoXtsMover := MoverInterface;
END_METHOD

END_FUNCTION_BLOCK

// ---- Tasks/ActivateTrackForMover.TcPOU
FUNCTION_BLOCK ActivateTrackForMover EXTENDS TaskBase
VAR_INPUT
END_VAR
VAR_OUTPUT
END_VAR
VAR
	mcActivateTrack : Tc3_McCollisionAvoidance.MC_ActivateTrack;
	_axis : REFERENCE TO Tc2_MC2.AXIS_REF;
	_ActivateTrack : BOOL;
	_newTrackId : OTCID;
END_VAR

METHOD Abort : BOOL
mcActivateTrack.Execute := FALSE;
_busy := FALSE;
_ActivateTrack := FALSE;
Abort := TRUE;
State := 0;
END_METHOD

METHOD Cycle : BOOL
VAR_INPUT
END_VAR
CASE State OF
	0:
		IF _ActivateTrack THEN
			_done := FALSE;
			_error := FALSE;
			_busy := TRUE;
			mcActivateTrack.Execute := TRUE;
			IF mcActivateTrack.Busy THEN
				State := 10;
				_ActivateTrack := FALSE;
			END_IF
		END_IF
	
	10:
		IF NOT mcActivateTrack.Busy THEN
			IF mcActivateTrack.Done THEN
				_done := TRUE;
				_newTrackId := mcActivateTrack.TrackId;
			ELSIF mcActivateTrack.Error THEN
				_error := TRUE;
			END_IF
			_busy := FALSE;
			mcActivateTrack.Execute := FALSE;
			State := 0;
		END_IF
END_CASE

mcActivateTrack(Axis := _axis);
END_METHOD

METHOD PUBLIC Execute : BOOL
VAR_INPUT
	Track : OTCID;
END_VAR
Execute := _ActivateTrack := TRUE;
mcActivateTrack.TrackId := Track;
END_METHOD

METHOD FB_init : BOOL
VAR_INPUT
	bInitRetains : BOOL; // if TRUE, the retain variables are initialized (warm start / cold start)
	bInCopyCode : BOOL;  // if TRUE, the instance afterwards gets moved into the copy code (online change)
	axis : reference TO AXIS_REF;
END_VAR
_axis REF= axis;
END_METHOD

PROPERTY PUBLIC NewTrackId : OTCID
GET
NewTrackId := _newTrackId;
END_GET
END_PROPERTY

END_FUNCTION_BLOCK

// ---- Tasks/MoveModuloMoverToPosition.TcPOU
FUNCTION_BLOCK MoveModuloMoverToPosition EXTENDS TaskBase
VAR_INPUT
END_VAR
VAR_OUTPUT
END_VAR
VAR
	moveAbs	: MC_MoveAbsoluteCA;
	_axis : REFERENCE TO AXIS_REF;
	_MoveMover : BOOL;
	_stOptions : ST_MoveAbsoluteCAOptions;
END_VAR

METHOD Abort : BOOL
moveAbs.Execute := FALSE;
moveAbs.Position := moveAbs.Velocity := 0;
_MoveMover := false;
_busy := false;
Abort := true;
State := 0;
END_METHOD

PROPERTY PUBLIC Acceleration : mc_lreal
GET
Acceleration := moveAbs.Acceleration;
END_GET
SET
moveAbs.Acceleration := Acceleration;
END_SET
END_PROPERTY

METHOD Cycle : BOOL
VAR_INPUT
END_VAR
CASE State OF
	0:
		IF _MoveMover THEN
			_done := FALSE;
			_error := FALSE;
			_busy := TRUE;
			moveAbs.Execute := TRUE;
			IF moveAbs.Busy THEN
				State := 10;
				_MoveMover := FALSE;
			END_IF
		END_IF
		
	10:
		IF NOT moveAbs.Busy THEN
			IF moveAbs.Done THEN
				_done := TRUE;
			ELSIF moveAbs.Error THEN
				_error := TRUE;
			END_IF
			_busy := FALSE;
			moveAbs.Execute := FALSE;
			State := 0;
		END_IF
END_CASE

moveAbs(Axis := _axis, Options := _stOptions);
END_METHOD

PROPERTY PUBLIC Deceleration : mc_lreal
GET
Deceleration := moveAbs.Deceleration;
END_GET
SET
moveAbs.Deceleration := Deceleration;
END_SET
END_PROPERTY

METHOD FB_init : BOOL
VAR_INPUT
	bInitRetains : BOOL; // if TRUE, the retain variables are initialized (warm start / cold start)
	bInCopyCode : BOOL;  // if TRUE, the instance afterwards gets moved into the copy code (online change)
	axis : reference TO AXIS_REF;
END_VAR
_axis REF= axis;
END_METHOD

PROPERTY PUBLIC Gap : mc_lreal
GET
Gap := moveAbs.Gap;
END_GET
SET
moveAbs.Gap := Gap;
END_SET
END_PROPERTY

PROPERTY PUBLIC Jerk : mc_lreal
GET
Jerk := moveAbs.Jerk;
END_GET
SET
moveAbs.Jerk := Jerk;
END_SET
END_PROPERTY

METHOD MoveTo : BOOL
VAR_INPUT
	Position : MC_LREAL;
	Velocity : MC_LREAL;
	Direction: Tc3_Mc3Definitions.MC_DIRECTION;
	Turns: UDINT;
END_VAR
moveAbs.Position := Position;
moveAbs.Velocity := Velocity;
moveAbs.Direction := Direction;
moveAbs.Options.AdditionalTurns := Turns;
_MoveMover := MoveTo := true;
END_METHOD

PROPERTY PUBLIC Options : ST_MoveAbsoluteCAOptions
GET
Options := _stOptions;
END_GET
SET
_stOptions := Options;
END_SET
END_PROPERTY

END_FUNCTION_BLOCK

// ---- PackML/PMLStateMachine.TcPOU
FUNCTION_BLOCK PMLStateMachine EXTENDS CyclicBase IMPLEMENTS IPmlStateMachine
VAR_INPUT
END_VAR
VAR_OUTPUT
END_VAR
VAR
	_pmlStateMachine : Tc3_PackML_V2.PML_StateMachine;
	_pmlModeMachine : Tc3_PackML_V2.PML_UnitModeManager;
	_subUnits : ARRAY[0..9] OF IPmlStateMachine;
	subUnitArray : ARRAY[0..9] OF ST_PMLSubUnitInfo;
	_SubUnitReference: ST_PMLSubUnitInfoRef;
	modeChangeTrigger : Tc2_Standard.R_TRIG;
	i: DINT;
END_VAR

METHOD PUBLIC  Cycle : BOOL
VAR_INPUT
END_VAR
IF _SubUnitReference.NoOfSubUnits <> 0 THEN
	FOR i := 0 TO 9 DO
		IF _subUnits[i] <> 0 THEN
			subUnitArray[i].eState := _subUnits[i].GetCurrentState();
			subUnitArray[i].Active := True;
		END_IF
	END_FOR
	_SubUnitReference.pArray := ADR(subUnitArray);
	_SubUnitReference.ArraySize := SIZEOF(subUnitArray);
END_IF

_pmlStateMachine(eMode := _pmlModeMachine.eModeStatus, stSubUnitInfoRef := _SubUnitReference);
_pmlModeMachine(eState := _pmlStateMachine.eState, bExecute := modeChangeTrigger.Q);
modeChangeTrigger();
END_METHOD

METHOD PUBLIC GetCurrentMode : E_PmlProtectedUnitMode
VAR_INPUT
END_VAR
GetCurrentMode := _pmlModeMachine.eModeStatus;
END_METHOD

METHOD PUBLIC GetCurrentState : E_PMLState
VAR_INPUT
END_VAR
GetCurrentState := _pmlStateMachine.eState;
END_METHOD

METHOD PUBLIC PmlModeCommand : Bool
VAR_INPUT
	Mode : E_PMLProtectedUnitMode;
END_VAR
_pmlModeMachine.eModeCommand := Mode;
modeChangeTrigger.CLK := true;
END_METHOD

METHOD PUBLIC PmlStateCommand : BOOL
VAR_INPUT
	Command : E_PMLCommand;
END_VAR
_pmlStateMachine.eCommand := Command;
END_METHOD

METHOD PUBLIC RegisterSubUnit : IPmlStateMachine
VAR_INPUT
	SubUnit : IPmlStateMachine;
END_VAR
FOR i := 0 TO 9 DO
	IF _subUnits[i] = 0 THEN
		_subUnits[i] := SubUnit;
		_SubUnitReference.NoOfSubUnits := i + 1;
		EXIT;
	END_IF
END_FOR
END_METHOD

METHOD PUBLIC SetStateComplete : BOOL
VAR_INPUT
END_VAR
_pmlStateMachine.M_StateComplete();
END_METHOD

END_FUNCTION_BLOCK

// ---- SequenceSamples/IndexMoverSequence.TcPOU
FUNCTION_BLOCK IndexMoverSequence EXTENDS CyclicBase
VAR
	State : IndexSequenceState;  
	CurrentStation : INT;
	TargetStationPosition : MC_LREAL;
	_MoverVelocity : MC_LREAL := 1000.0;
	stSequenceInfo : MoverSequenceInfo;
	StationArray : ARRAY[1..SystemParameters.NumberOfStations] OF IProcess;
	ThisMover : IMover;
	XtsTrack : IXtsTrack;
	StateMachine : IPmlStateMachine;
END_VAR

METHOD Abort : BOOL
VAR_INPUT
END_VAR
State := IndexSequenceState.Available;
CurrentStation := 0;
TargetStationPosition := 0.0;
stSequenceInfo.CurrentStation := CurrentStation;
stSequenceInfo.MoverId := ThisMover.AxisRef.NcToPlc.AxisId;
stSequenceInfo.State := State;
stSequenceInfo.Velocity := ThisMover.AxisRef.NcToPlc.ActVelo;
END_METHOD

METHOD PUBLIC  Cycle : BOOL
VAR_INPUT
END_VAR
IF StateMachine.GetCurrentState() = E_PMLState.ePMLState_Aborting THEN
	State := IndexSequenceState.Aborting;
ELSIF StateMachine.GetCurrentState() = E_PMLState.ePMLState_Stopping THEN
	State := IndexSequenceState.Stopping;
END_IF
CASE State OF
	IndexSequenceState.Init:
		IF ThisMover.isDetected() THEN
			State := IndexSequenceState.Available;
		END_IF
		
	IndexSequenceState.Available:
		IF StateMachine.GetCurrentState() = E_PMLState.ePMLState_Execute THEN
			State := IndexSequenceState.MovingToStart;
		END_IF
		
	IndexSequenceState.MovingToStart:
		IF ThisMover.isAtPosition(position := XtsTrack.HomePosition) THEN
			State := IndexSequenceState.AtStart;
		END_IF
			
	IndexSequenceState.AtStart:
		IF StationArray[1].IsReady() THEN
			State := IndexSequenceState.GetNextMove;
		END_IF

	IndexSequenceState.MovingToStation:
		IF ThisMover.isStationary() THEN 
			IF ThisMover.isAtPosition(TargetStationPosition) THEN
				IF StationArray[CurrentStation].IsProcess THEN
					State := IndexSequenceState.AtProcess;
				ELSE
					State := IndexSequenceState.AtStation;
				END_IF
				StationArray[CurrentStation].HasMover(ThisMover);
			ELSE
				State := IndexSequenceState.QueuedAtStation;
			END_IF
		END_IF
		
	IndexSequenceState.QueuedAtStation:
		IF NOT ThisMover.isStationary() THEN
				State := IndexSequenceState.MovingToStation;
		END_IF

	IndexSequenceState.AtStation:
		IF StationArray[CurrentStation].isComplete() THEN
			State := IndexSequenceState.GetNextMove;
		END_IF

	IndexSequenceState.AtProcess:
		ThisMover.MoveTo(Position := StationArray[CurrentStation].EndPosition,
								Velocity := StationArray[CurrentStation].ProcessVelocity,
								BackwardMove := FALSE);
		State := IndexSequenceState.InProcess;
								
	IndexSequenceState.InProcess:
		IF ThisMover.isStationary() THEN 
			IF ThisMover.isAtPosition(StationArray[CurrentStation].EndPosition) THEN
				State := IndexSequenceState.GetNextMove;
			END_IF
		END_IF
	
	IndexSequenceState.GetNextMove:
		IF CurrentStation = SystemParameters.NumberOfStations THEN
			IF ThisMover.MoveTo(Position := XtsTrack.HomePosition,
							Velocity := _MoverVelocity,
							BackwardMove := FALSE) THEN
				State := IndexSequenceState.MovingToStart;
				StationArray[CurrentStation].MoverAway();
				CurrentStation := 0; 
			END_IF
		ELSE
			State := IndexSequenceState.GoToNextStation;
		END_IF
		
	IndexSequenceState.GoToNextStation:
		IF StationArray[CurrentStation + 1].IsProcess THEN
			TargetStationPosition := StationArray[CurrentStation + 1].StartPosition;
		ELSE
			TargetStationPosition := StationArray[CurrentStation + 1].Position;
		END_IF
		IF 	ThisMover.MoveTo(Position := TargetStationPosition,
							Velocity := _MoverVelocity,
							BackwardMove := FALSE) THEN
			IF CurrentStation <> 0 THEN
				StationArray[CurrentStation].MoverAway();	
			END_IF		
			CurrentStation := CurrentStation + 1;
			State := IndexSequenceState.MovingToStation;
		END_IF	

	IndexSequenceState.Stopping:
		IF StateMachine.GetCurrentState() = E_PMLState.ePMLState_Stopped THEN
			State := IndexSequenceState.Available;
			CurrentStation := 0;
			TargetStationPosition := 0.0;
		END_IF			
		
	IndexSequenceState.Aborting:
		IF StateMachine.GetCurrentState() = E_PMLState.ePMLState_Aborted THEN
			State := IndexSequenceState.Available;
			CurrentStation := 0;
			TargetStationPosition := 0.0;
		END_IF
END_CASE

//Cyclic update info data
stSequenceInfo.CurrentStation := CurrentStation;
stSequenceInfo.MoverId := ThisMover.AxisRef.NcToPlc.AxisId;
stSequenceInfo.State := State;
stSequenceInfo.Velocity := ThisMover.AxisRef.NcToPlc.ActVelo;
END_METHOD

PROPERTY MoverVelocity : mc_lreal
GET
MoverVelocity := _MoverVelocity;
END_GET
SET
_MoverVelocity := MoverVelocity;
END_SET
END_PROPERTY

PROPERTY MyMover : IMover
GET
MyMover := ThisMover;
END_GET
SET
ThisMover := MyMover;
END_SET
END_PROPERTY

PROPERTY MyStations : ARRAY[1..SystemParameters.NumberOfStations] OF IProcess
GET
MyStations := StationArray;
END_GET
SET
StationArray := MyStations;
END_SET
END_PROPERTY

PROPERTY PmlStateMachine : IPmlStateMachine
GET
PmlStateMachine := StateMachine;
END_GET
SET
StateMachine := PmlStateMachine;
END_SET
END_PROPERTY

PROPERTY XtsTrackController : IXtsTrack
GET
XtsTrackController := XtsTrack;
END_GET
SET
XtsTrack := XtsTrackController;
END_SET
END_PROPERTY

END_FUNCTION_BLOCK

// ---- Station Class/Process/Process.TcPOU
FUNCTION_BLOCK Process EXTENDS Station IMPLEMENTS IProcess
VAR_INPUT
END_VAR
VAR_OUTPUT
END_VAR
VAR
	_isProcess : BOOL;
	_startPos : MC_LREAL;
	_endPos : MC_LREAL;
	_processVelo : MC_LREAL;
END_VAR

METHOD PUBLIC  Cycle : BOOL
VAR_INPUT
END_VAR
SUPER^.Cycle();
END_METHOD

PROPERTY EndPosition : MC_LREAL
GET
EndPosition := _endPos;
END_GET
SET
_endPos := EndPosition;
END_SET
END_PROPERTY

PROPERTY IsProcess : BOOL
GET
IsProcess := _isProcess;
END_GET
SET
_isProcess := IsProcess;
END_SET
END_PROPERTY

PROPERTY ProcessVelocity : MC_LREAL
GET
ProcessVelocity := _processVelo;
END_GET
SET
_processVelo := ProcessVelocity;
END_SET
END_PROPERTY

PROPERTY StartPosition : MC_LREAL
GET
StartPosition := _startPos;
END_GET
SET
_startPos := StartPosition;
END_SET
END_PROPERTY

END_FUNCTION_BLOCK

// ---- Station Class/Station/Station.TcPOU
FUNCTION_BLOCK Station EXTENDS CyclicBase IMPLEMENTS IStation
VAR_INPUT
END_VAR
VAR_OUTPUT
END_VAR
VAR
	_Clear : BOOL;
	_Complete : BOOL;
	_Operating : BOOL;
	_Ready : BOOL;
	_Positions : ARRAY[1..4] OF MC_LREAL := [0.0,0.0,0.0,0.0];
	NumberOfPositions : INT := 0;
	AssignedPositions : INT := 1;
	StationMovers : INT;
	stInfo : stStationInfo;
	_HasMover : BOOL;
	ProductCounter : R_TRIG;
	Products : DINT;
	LastStation : BOOL;
	MyMover : IMover;
END_VAR

METHOD Abort : BOOL
VAR_INPUT
END_VAR
_Complete := FALSE;
_Clear := TRUE;
_Operating := FALSE;
_Ready := TRUE;
END_METHOD

METHOD PUBLIC  Cycle : BOOL
VAR_INPUT
END_VAR
//Cyclic info
stInfo.StationPosition := _Positions[1];
stInfo.StationStatus.Clear := _clear;
stInfo.StationStatus.Complete := _Complete;
stInfo.StationStatus.HasMover := _HasMover;
stInfo.StationStatus.Operating := _Operating;
stInfo.StationStatus.Ready := _Ready;

IF LastStation THEN
	ProductCounter(CLK := _Complete);
	IF ProductCounter.Q THEN
		Products := Products + 1;
	END_IF
END_IF
END_METHOD

METHOD HasMover : BOOL
VAR_INPUT
	mover : IMover;
END_VAR
StationMovers := StationMovers + 1;
IF StationMovers = NumberOfPositions THEN
	_HasMover := TRUE;
END_IF
MyMover := mover;
END_METHOD

METHOD IsClear : BOOL
IsClear := _Clear;
END_METHOD

METHOD isComplete : BOOL
isComplete := _Complete;
END_METHOD

PROPERTY PUBLIC IsLastStation : BOOL
GET
IsLastStation := LastStation;
END_GET
SET
LastStation := IsLastStation;
END_SET
END_PROPERTY

METHOD IsOperating : BOOL
IsOperating := _Operating;
END_METHOD

METHOD IsReady : BOOL
IsReady := _Ready;
END_METHOD

METHOD MoverAway : BOOL
VAR_INPUT
END_VAR
StationMovers := StationMovers - 1;
MyMover := 0;
END_METHOD

PROPERTY Position : MC_LREAL
GET
Position := _Positions[AssignedPositions];
AssignedPositions := AssignedPositions + 1;
IF AssignedPositions > NumberOfPositions THEN
	AssignedPositions := 1;
END_IF
END_GET
SET
IF NumberOfPositions < 5 THEN
	NumberOfPositions := NumberOfPositions + 1;
	_Positions[NumberOfPositions] := Position;
END_IF
END_SET
END_PROPERTY

END_FUNCTION_BLOCK

// ---- Station Class/Station/StationSample.TcPOU
FUNCTION_BLOCK StationSample EXTENDS Process
VAR
	_OperationTime : TIME := T#1S;
	Operation : ton;
	State: INT;
	StateMachine : IPmlStateMachine;
END_VAR

METHOD Abort : BOOL
VAR_INPUT
END_VAR
SUPER^();
StationMovers := State := 0;
END_METHOD

METHOD Cycle : BOOL
VAR_INPUT
END_VAR
IF _isProcess THEN
	;
ELSE
	CASE State OF
		0:
			IF _HasMover THEN
				_Operating := TRUE;
				_Clear := FALSE;
				_Ready := FALSE;
				Operation.IN := TRUE;
				State := 1;
			END_IF
		1:
			IF Operation.Q THEN
				_Complete := TRUE;
				IF StationMovers = 0 THEN
					_HasMover := FALSE;
					Operation.IN := FALSE;
				END_IF
				State := 2;
			END_IF
		2:
			_Complete := FALSE;
			_Clear := TRUE;
			_Operating := FALSE;
			_Ready := TRUE;
			State := 0;
	END_CASE	
	Operation(PT := _OperationTime);
END_IF

IF StateMachine.GetCurrentState() = E_PMLState.ePMLState_Aborted 
	OR StateMachine.GetCurrentState() = E_PMLState.ePMLState_Stopping THEN
	_Complete := FALSE;
	_Clear := TRUE;
	_Operating := FALSE;
	_Ready := TRUE;
	StationMovers := State := 0;
END_IF

SUPER^.Cycle();
stInfo.StationProcessTime := _OperationTime;
END_METHOD

PROPERTY PmlStateMachine : IPmlStateMachine
GET
PmlStateMachine := StateMachine;
END_GET
SET
StateMachine := PmlStateMachine;
END_SET
END_PROPERTY

PROPERTY TempPropTime : time
GET
TempPropTime := _OperationTime;
END_GET
SET
_OperationTime := TempPropTime;
END_SET
END_PROPERTY

END_FUNCTION_BLOCK

// ---- Station Class/TMSStation/TmsEmbarkStation.TcPOU
FUNCTION_BLOCK TmsEmbarkStation EXTENDS Process IMPLEMENTS ITF_SwitchStation
VAR_INPUT
	StateMachine : IPmlStateMachine;
	TmsSwitch : ITF_TmsSwitch;
END_VAR
VAR_OUTPUT
END_VAR
VAR
	DepartMover : ITmsMover;
	_TrackLevel : INT := 1; //1 is low, 2 is high
	State :(
		Init,                                               
		Ready,                                 
        Waiting,
		HasSwitch,
		Call,
		Processing,
		Boarding,
		BoardingComplete,
		Moving,
		Aborting); 
	_switchPosition: MC_LREAL;
	demandPosition : TmsSwitchPosition;
	arrTrackIds : ARRAY[1..4] OF OTCID;
	isUpAllowed : BOOL := TRUE;
	isDownAllowed : BOOL := FALSE;
	isMiddleAllowed : BOOL := TRUE;
	BoardVelocity : MC_LREAL := 100.0;
END_VAR

METHOD PUBLIC  Cycle : BOOL
VAR_INPUT
END_VAR
CASE State OF
	Init:
		_Operating := _Clear := _Complete := _Ready := _HasMover := FALSE;
		StationMovers := 0;
		State := Ready;
	
	Ready:	
		IF StateMachine.GetCurrentState() = E_PMLState.ePMLState_Clearing THEN
			_Operating := _Complete := _HasMover := FALSE;
			_Clear := _Ready := TRUE;
			StationMovers := 0;
			State := Waiting;
		END_IF
		IF StateMachine.GetCurrentState() = E_PMLState.ePMLState_Aborting THEN
			State := Aborting;
		END_IF
	
	Waiting:
		IF _HasMover THEN
			State := HasSwitch;
			_Operating := TRUE;
			_Clear := FALSE;
			_Ready := FALSE;
			_Complete := FALSE;
		END_IF
		IF StateMachine.GetCurrentState() = E_PMLState.ePMLState_Aborting THEN
			State := Aborting;
		END_IF
	
	HasSwitch:
		IF (_TrackLevel = 1 AND (TmsSwitch.Switch = TmsSwitchPosition.Down OR (TmsSwitch.Switch = TmsSwitchPosition.Middle AND isUpAllowed)))
			OR (_TrackLevel = 2 AND (TmsSwitch.Switch = TmsSwitchPosition.Up OR (TmsSwitch.Switch = TmsSwitchPosition.Middle AND isDownAllowed))) THEN
				IF TmsSwitch.ExchangeMover(Mover := DepartMover, currentStation := THIS^) THEN
					State := Processing;
				END_IF
		ELSE
			State := Call;
		END_IF
		IF StateMachine.GetCurrentState() = E_PMLState.ePMLState_Aborting THEN
			State := Aborting;
		END_IF	
		
	Call:
		IF NOT TmsSwitch.HasMover() AND TmsSwitch.IsStationary() THEN
			IF TmsSwitch.MoveTo(positionState := TmsSwitchPosition.Middle) THEN
				State := HasSwitch;
			END_IF
		ELSE
			State := Waiting;
		END_IF
		IF StateMachine.GetCurrentState() = E_PMLState.ePMLState_Aborting THEN
			State := Aborting;
		END_IF
	
	Processing:
		IF _TrackLevel = 1 THEN
			IF TmsSwitch.Switch = TmsSwitchPosition.Down and isMiddleAllowed THEN
				IF DepartMover.ActiveTrack = arrTrackIds[4] THEN
					State := Boarding;
				ELSE
					DepartMover.ActivateTrack(arrTrackIds[4]);
					State := Boarding;
				END_IF
				demandPosition := TmsSwitchPosition.Middle;
			ELSIF TmsSwitch.Switch = TmsSwitchPosition.Middle AND isUpAllowed THEN
				IF DepartMover.ActiveTrack = arrTrackIds[1] THEN
					State := Boarding;
				ELSE
					DepartMover.ActivateTrack(arrTrackIds[1]);
					State := Boarding;
				END_IF
				demandPosition := TmsSwitchPosition.Up;
			END_IF
		ELSE
			IF TmsSwitch.Switch = TmsSwitchPosition.Up AND isMiddleAllowed THEN
				IF DepartMover.ActiveTrack = arrTrackIds[3] THEN
					State := Boarding;
				ELSE
					DepartMover.ActivateTrack(arrTrackIds[3]);
					State := Boarding;
				END_IF
				demandPosition := TmsSwitchPosition.Middle;
			ELSIF TmsSwitch.Switch = TmsSwitchPosition.Middle AND isDownAllowed THEN
				IF DepartMover.ActiveTrack = arrTrackIds[2] THEN
					State := Boarding;
				ELSE
					DepartMover.ActivateTrack(arrTrackIds[2]);
					State := Boarding;
				END_IF
				demandPosition := TmsSwitchPosition.Down;
			END_IF
		END_IF
		IF StateMachine.GetCurrentState() = E_PMLState.ePMLState_Aborting THEN
			State := Aborting;
		END_IF
		
	Boarding:
		DepartMover.MoveTo(Position := _switchPosition, Velocity := BoardVelocity, BackwardMove := FALSE);
		IF DepartMover.isAtPosition(position := _switchPosition) THEN
			State := BoardingComplete;
		END_IF
		
	BoardingComplete:
		IF TmsSwitch.MoveTo(positionState := demandPosition) THEN
			State := Moving;
		END_IF
		IF StateMachine.GetCurrentState() = E_PMLState.ePMLState_Aborting THEN
			State := Aborting;
		END_IF
		
	Moving:
		IF _Complete AND NOT _HasMover THEN
			_Operating := FALSE;
			_Clear := TRUE;
			_Ready := TRUE;
			State := Waiting;
		END_IF
		IF StateMachine.GetCurrentState() = E_PMLState.ePMLState_Aborting THEN
			State := Aborting;
		END_IF	

	Aborting:
		State := Ready;	
		DepartMover := 0;
END_CASE
SUPER^.Cycle();
END_METHOD

METHOD HasMover : BOOL
VAR_INPUT
	mover : IMover;
END_VAR
VAR
	iTmsMover : ITmsMover;
END_VAR
IF StationMovers <= 2 THEN
	StationMovers := StationMovers + 1;
	IF __QUERYINTERFACE(mover,iTmsMover) THEN
		DepartMover := iTmsMover;
		_HasMover := true;
	END_IF
END_IF
END_METHOD

METHOD PUBLIC MoverAway : BOOL
VAR_INPUT
END_VAR
StationMovers := StationMovers - 1;
IF StationMovers = 0 THEN
	_HasMover := FALSE;
END_IF
DepartMover := 0;
END_METHOD

METHOD PUBLIC SwitchMoveComplete : BOOL
VAR_INPUT
END_VAR
_Complete := SwitchMoveComplete := true;
END_METHOD

PROPERTY SwitchTravelPosition : mc_lreal
GET
SwitchTravelPosition := _switchPosition;
END_GET
SET
_switchPosition := SwitchTravelPosition;
END_SET
END_PROPERTY

PROPERTY TrackIds : array[1..4] of otcid
GET
TrackIds := arrTrackIds;
END_GET
SET
arrTrackIds := TrackIds;
END_SET
END_PROPERTY

PROPERTY TrackLevel : INT
GET
TrackLevel := _TrackLevel;
END_GET
SET
_TrackLevel := TrackLevel;
END_SET
END_PROPERTY

END_FUNCTION_BLOCK

// ---- Station Class/TMSStation/TmsExchange.TcPOU
FUNCTION_BLOCK PUBLIC TmsExchange EXTENDS Process
VAR_INPUT
	TmsSwitch : ITF_TmsSwitch;
	StateMachine : IPmlStateMachine;
END_VAR
VAR_OUTPUT
END_VAR
VAR
	holdingStation : TmsHoldStation;
	embarkingStation : TmsEmbarkStation;
END_VAR

holdingStation(StateMachine := StateMachine, embarkStation := embarkingStation);
embarkingStation(StateMachine := StateMachine, TmsSwitch := TmsSwitch);

PROPERTY EmbarkStation : IProcess
GET
EmbarkStation := embarkingStation;
END_GET
END_PROPERTY

PROPERTY ExchangeTrackLevel : int
GET
ExchangeTrackLevel := embarkingStation.TrackLevel;
END_GET
SET
embarkingStation.TrackLevel := ExchangeTrackLevel;
END_SET
END_PROPERTY

PROPERTY HoldStation : IProcess
GET
HoldStation := holdingStation;
END_GET
END_PROPERTY

PROPERTY SwitchTravelPosition : MC_LREAL
GET
SwitchTravelPosition := embarkingStation.SwitchTravelPosition;
END_GET
SET
embarkingStation.SwitchTravelPosition := SwitchTravelPosition;
END_SET
END_PROPERTY

PROPERTY PUBLIC TrackIds : Array[1..4] of OTCID
GET
TrackIds := embarkingStation.TrackIds;
END_GET
SET
embarkingStation.TrackIds := TrackIds;
END_SET
END_PROPERTY

END_FUNCTION_BLOCK

// ---- Station Class/TMSStation/TmsHoldStation.TcPOU
FUNCTION_BLOCK TmsHoldStation EXTENDS Process 
VAR_INPUT
	StateMachine : IPmlStateMachine;
	embarkStation : IProcess;
END_VAR
VAR_OUTPUT
END_VAR
VAR
	HoldMover : ITmsMover;
	State :(
		Init,                                               
		Ready,                                 
        Waiting,
		Processing,
		Clearing,
		Aborting); 
END_VAR

METHOD PUBLIC  Cycle : BOOL
VAR_INPUT
END_VAR
CASE State OF
	Init:
		_Operating := _Clear := _Complete := _Ready := _HasMover := FALSE;
		StationMovers := 0;
		State := Ready;
	
	Ready:	
		IF StateMachine.GetCurrentState() = E_PMLState.ePMLState_Clearing THEN
			_Operating := _Complete := _HasMover := FALSE;
			_Clear := _Ready := TRUE;
			StationMovers := 0;
			State := Waiting;
		END_IF
		IF StateMachine.GetCurrentState() = E_PMLState.ePMLState_Aborting THEN
			State := Aborting;
		END_IF
	
	Waiting:
		IF _HasMover THEN
			State := Processing;
			_Operating := TRUE;
			_Clear := FALSE;
			_Ready := FALSE;
		END_IF
		IF StateMachine.GetCurrentState() = E_PMLState.ePMLState_Aborting THEN
			State := Aborting;
		END_IF
		
	Processing:
		IF embarkStation.IsClear() THEN
			_Complete := TRUE;
			State := Clearing;
		END_IF
		IF StateMachine.GetCurrentState() = E_PMLState.ePMLState_Aborting THEN
			State := Aborting;
		END_IF
		
	Clearing:
		State := Waiting;
		_Operating := FALSE;
		_Clear := TRUE;
		_Ready := TRUE;
		_Complete := FALSE;
		HoldMover := 0;
		
	Aborting:
		State := Ready;
		HoldMover := 0;
		_HasMover := FALSE;
END_CASE
SUPER^.Cycle();
END_METHOD

METHOD HasMover : BOOL
VAR_INPUT
	mover : IMover;
END_VAR
VAR
	iTmsMover : ITmsMover;
END_VAR
IF StationMovers <= 2 THEN
	StationMovers := StationMovers + 1;
	IF __QUERYINTERFACE(mover,iTmsMover) THEN
		HoldMover := iTmsMover;
		_HasMover := TRUE;
	END_IF
END_IF
END_METHOD

METHOD PUBLIC MoverAway : BOOL
VAR_INPUT
END_VAR
StationMovers := StationMovers - 1;
IF StationMovers = 0 THEN
	_HasMover := FALSE;
END_IF
HoldMover := 0;
END_METHOD

END_FUNCTION_BLOCK

// ---- Switch Class/DualModuleTmsSwitch.TcPOU
FUNCTION_BLOCK DualModuleTmsSwitch EXTENDS MC2_Axis_Base IMPLEMENTS ITF_TmsSwitch
VAR_INPUT
	StateMachine : IPmlStateMachine;
END_VAR
VAR_OUTPUT
END_VAR
VAR
	_exchangeMover : IMover;
	_currentStation : ITF_SwitchStation;
	_demandPosition : MC_LREAL;
	_upPosition : MC_LREAL;
	_middlePosition : MC_LREAL;
	_downPosition : MC_LREAL;
	SwitchVelocity : MC_LREAL := 100.0;
	arrTrackIds : ARRAY[1..4] OF OTCID;
	stSwitchInfo : TmsSwitchInfo;
END_VAR

METHOD Cycle : BOOL
VAR_INPUT
END_VAR
CASE stSwitchInfo.State OF
	TmsSwitchState.Init:
		IF NOT THIS^.hasError() THEN
			stSwitchInfo.State := TmsSwitchState.Ready;
		END_IF
		
	TmsSwitchState.Ready:
		IF StateMachine.GetCurrentState() = E_PMLState.ePMLState_Clearing THEN
			SUPER^.EnableAxis();
			stSwitchInfo.State := TmsSwitchState.Enabling;
		END_IF	
		
	TmsSwitchState.Enabling:
		IF SUPER^.isEnabled() THEN
			stSwitchInfo.State := TmsSwitchState.Enabled;
		END_IF
		
	TmsSwitchState.Enabled:
		IF StateMachine.GetCurrentState() = E_PMLState.ePMLState_Resetting THEN
			IF SUPER^.MoveToPosition(Position := _middlePosition, Velocity := 100.0) OR SUPER^.isAtPosition(position := _middlePosition) THEN
				stSwitchInfo.State := TmsSwitchState.Resetting;
			END_IF
		END_IF
		IF StateMachine.GetCurrentState() = E_PMLState.ePMLState_Aborting
			OR StateMachine.GetCurrentState() = E_PMLState.ePMLState_Stopping THEN
			SUPER^.DisableAxis();
			stSwitchInfo.State := TmsSwitchState.Disabling;
		END_IF
		
	TmsSwitchState.Resetting:
		IF SUPER^.isAtPosition(position := MiddlePosition) THEN
			stSwitchInfo.State := TmsSwitchState.Waiting;
		END_IF	
	
	TmsSwitchState.Waiting:
		IF StateMachine.GetCurrentState() = E_PMLState.ePMLState_Aborting
			OR StateMachine.GetCurrentState() = E_PMLState.ePMLState_Stopping THEN
			SUPER^.DisableAxis();
			stSwitchInfo.State := TmsSwitchState.Disabling;
		END_IF
		
	TmsSwitchState.AssignMover:
		IF HasMover() THEN
			IF FindNewTrack() <> 0 THEN
				stSwitchInfo.State := TmsSwitchState.Moving;
			END_IF
		ELSE
			stSwitchInfo.State := TmsSwitchState.Moving;
		END_IF

	TmsSwitchState.Moving:	
		IF SUPER^.isAtPosition(_demandPosition) THEN
			stSwitchInfo.State := TmsSwitchState.Done;
		END_IF
	
	TmsSwitchState.Done:
		IF _currentStation <> 0 THEN
			IF _currentStation.SwitchMoveComplete() THEN
				_exchangeMover := 0;
				_currentStation := 0;
			END_IF	
		END_IF
		stSwitchInfo.State := TmsSwitchState.Waiting;

	TmsSwitchState.Disabling:
		IF NOT THIS^.isEnabled() THEN
			THIS^.ResetAxis();
			stSwitchInfo.State := TmsSwitchState.Init;
		END_IF

END_CASE

//Cyclic get switch info
stSwitchInfo.ActPos := SUPER^._axis.NcToPlc.ActPos;
stSwitchInfo.Position := Switch;

SUPER^.Cycle();
END_METHOD

PROPERTY DownPosition : MC_LREAL
GET
DownPosition := _downPosition;
END_GET
SET
_downPosition := DownPosition;
END_SET
END_PROPERTY

METHOD PUBLIC ExchangeMover : BOOL
VAR_INPUT
	Mover : IMover;
	CurrentStation : ITF_SwitchStation;
END_VAR
IF _exchangeMover = 0 AND stSwitchInfo.State = TmsSwitchState.Waiting AND NOT (stSwitchInfo.Mode = TmsSwitchMode.Manual) THEN
	_exchangeMover := Mover;	
	_currentStation := CurrentStation;
	ExchangeMover := TRUE;
END_IF
END_METHOD

METHOD PUBLIC FindNewTrack : OTCID
VAR_INPUT
END_VAR
VAR
	iTmsMover : ITmsMover;
END_VAR
IF __QUERYINTERFACE(_exchangeMover,iTmsMover) THEN
	IF Switch = TmsSwitchPosition.Up THEN
		IF iTmsMover.ActiveTrack = arrTrackIds[3] THEN
			iTmsMover.ActivateTrack(newTrack := arrTrackIds[1]);
		END_IF
	ELSIF Switch = TmsSwitchPosition.Middle THEN
		IF iTmsMover.ActiveTrack = arrTrackIds[1] THEN
			iTmsMover.ActivateTrack(newTrack := arrTrackIds[3]);
		ELSIF iTmsMover.ActiveTrack = arrTrackIds[2] THEN
			iTmsMover.ActivateTrack(newTrack := arrTrackIds[4]);
		END_IF
	ELSE
		IF iTmsMover.ActiveTrack = arrTrackIds[4] THEN
			iTmsMover.ActivateTrack(newTrack := arrTrackIds[2]);	
		END_IF
	END_IF
END_IF
FindNewTrack := iTmsMover.ActiveTrack;
END_METHOD

METHOD HasMover : BOOL
VAR_INPUT
END_VAR
HasMover := _exchangeMover <> 0;
END_METHOD

PROPERTY PUBLIC MiddlePosition : MC_LREAL
GET
MiddlePosition := _middlePosition;
END_GET
SET
_middlePosition := MiddlePosition;
END_SET
END_PROPERTY

METHOD PUBLIC MoveTo : BOOL
VAR_INPUT
	positionState : TmsSwitchPosition;
END_VAR
CASE positionState OF
	TmsSwitchPosition.Down:
		IF NOT SUPER^.isAtPosition(position := _downPosition) THEN
			IF SUPER^.MoveToPosition(Position := _downPosition, Velocity := SwitchVelocity) THEN
				MoveTo := TRUE;
				stSwitchInfo.State := TmsSwitchState.AssignMover;
				_demandPosition := _downPosition;
			END_IF
		END_IF	
	TmsSwitchPosition.Middle:
		IF NOT SUPER^.isAtPosition(position := _middlePosition) THEN
			IF SUPER^.MoveToPosition(Position := _middlePosition, Velocity := SwitchVelocity) THEN
				MoveTo := TRUE;
				stSwitchInfo.State := TmsSwitchState.AssignMover;
				_demandPosition := _middlePosition;
			END_IF
		END_IF	
	TmsSwitchPosition.Up:
		IF NOT SUPER^.isAtPosition(position := _upPosition) THEN
			IF SUPER^.MoveToPosition(Position := _upPosition, Velocity := SwitchVelocity) THEN
				MoveTo := TRUE;
				stSwitchInfo.State := TmsSwitchState.AssignMover;
				_demandPosition := _upPosition;
			END_IF
		END_IF	
END_CASE
END_METHOD

METHOD SetAutomaticMode : BOOL
VAR_INPUT
END_VAR
stSwitchInfo.Mode := TmsSwitchMode.Automatic;
END_METHOD

METHOD SetManualMode : BOOL
VAR_INPUT
END_VAR
stSwitchInfo.Mode := TmsSwitchMode.Manual;
END_METHOD

PROPERTY PUBLIC Switch : TmsSwitchPosition
GET
IF SUPER^.isAtPosition(position := _upPosition) THEN
	Switch := TmsSwitchPosition.Up;
ELSIF SUPER^.isAtPosition(position := _middlePosition) THEN
	Switch := TmsSwitchPosition.Middle;
ELSIF SUPER^.isAtPosition(position := _downPosition) THEN
	Switch := TmsSwitchPosition.Down;
ELSE
	Switch := TmsSwitchPosition.Moving;
END_IF
END_GET
END_PROPERTY

PROPERTY TrackIds : array[1..4] of otcid
GET
TrackIds := arrTrackIds;
END_GET
SET
arrTrackIds := TrackIds;
END_SET
END_PROPERTY

PROPERTY PUBLIC UpperPosition : MC_LREAL
GET
UpperPosition := _upPosition;
END_GET
SET
_upPosition := UpperPosition;
END_SET
END_PROPERTY

END_FUNCTION_BLOCK

// ---- Tasks/MoveMoverToPositionZoned.TcPOU
FUNCTION_BLOCK PUBLIC MoveMoverToPositionZoned EXTENDS MoveMoverToPosition
VAR_INPUT
END_VAR
VAR_OUTPUT
END_VAR
VAR
	StartZone: INT;
	CurrentZone : INT;
	ZoneTransitionPositions : ARRAY[1..4] OF DINT;
	ZoneVelocities : ARRAY[1..4] OF MC_LREAL;
END_VAR

METHOD Cycle : BOOL
VAR_INPUT
END_VAR
CASE State OF
	0:
		IF _MoveMover THEN
			_done := FALSE;
			_error := FALSE;
			_busy := TRUE;
			moveAbs.Execute := TRUE;
			StartZone := GetZone();
			moveAbs.Velocity := ZoneVelocities[StartZone];
			IF moveAbs.Busy THEN
				State := 10;
				_MoveMover := FALSE;
			END_IF
		END_IF
	
	10:
		IF NOT moveAbs.Busy THEN
			IF moveAbs.Done THEN
				_done := TRUE;
			ELSIF moveAbs.Error THEN
				_error := TRUE;
			END_IF
			_busy := FALSE;
			moveAbs.Execute := FALSE;
			State := 0;
		ELSE
			CurrentZone := GetZone();
			IF CurrentZone <> StartZone THEN
				moveAbs.Execute := FALSE;
				State := 0;
				_MoveMover := TRUE;
			END_IF
		END_IF
END_CASE

moveAbs(Axis := _axis);
END_METHOD

METHOD FB_init : BOOL
VAR_INPUT
	bInitRetains : BOOL; // if TRUE, the retain variables are initialized (warm start / cold start)
	bInCopyCode : BOOL;  // if TRUE, the instance afterwards gets moved into the copy code (online change)
	axis : REFERENCE TO AXIS_REF;
	arrPositions : ARRAY[1..4] OF DINT;
	arrVelos : ARRAY[1..4] OF MC_LREAL;
END_VAR
SUPER^();
ZoneTransitionPositions := arrPositions;
ZoneVelocities := arrVelos;
END_METHOD

METHOD GetZone : int
VAR_INPUT
END_VAR
IF _axis.NcToPlc.ModuloActPos > ZoneTransitionPositions[1] AND _axis.NcToPlc.ModuloActPos < ZoneTransitionPositions[2] THEN
	GetZone := 1;
ELSIF (_axis.NcToPlc.ModuloActPos > ZoneTransitionPositions[2] AND _axis.NcToPlc.ModuloActPos < 11000.0) 
		OR _axis.NcToPlc.ModuloActPos > 0.0 AND  _axis.NcToPlc.ModuloActPos < ZoneTransitionPositions[3] THEN
	GetZone := 2;
ELSIF _axis.NcToPlc.ModuloActPos > ZoneTransitionPositions[3] AND _axis.NcToPlc.ModuloActPos < ZoneTransitionPositions[4] THEN
	GetZone := 3;
ELSIF _axis.NcToPlc.ModuloActPos > ZoneTransitionPositions[4] THEN
	GetZone := 4;
ELSE
	GetZone := 4;
END_IF
END_METHOD

END_FUNCTION_BLOCK
